MailAddr := '"';
NbDest := 0;
FOR KK := 1 TO CstNbUser DO
	IF AX_Subscribed[KK] AND AX_MailAddr[KK] <> '' AND (AX_User_LVL[KK] AND Fifo.out.Alarms_LVL)>0 THEN		// If user is subscribed to this alarm, add his mail adress to the list. 
		IF MailAddr = '"' THEN
			MailAddr := concat('"', AX_MailAddr[KK]);	// Initialize first sender. 
		END_IF
		NbDest := NbDest + 1;
	END_IF
END_FOR

IF NbDest >0 THEN
	IF NbDest>1 THEN
		FOR KK := 1 TO CstNbUser DO
			IF AX_Subscribed[KK] AND MailAddr <> AX_MailAddr[KK] AND (AX_User_LVL[KK] AND Fifo.out.Alarms_LVL)>0 THEN
				MailAddr := concat(concat(MailAddr, ', '), AX_MailAddr[KK]);		// append other mail adress if several users subsribed to this alarm. 
			END_IF
		END_FOR
	END_IF
	MailAddr := concat(MailAddr, '" ');
	bSendMail := TRUE;
	bAlarmNoDestinator	:= FALSE;
ELSE 
	bAlarmNoDestinator	:= TRUE;
	bSendMail 			:= FALSE;

END_IF	

SendMail
(
	NETID := ParamNetID,
	PATHSTR := concat(IN_Directory, 'SMTP.exe'),
	DIRNAME := IN_Directory,
	COMNDLINE := concat(str1 := MailAddr, str2 := body),
	start := bSendMail AND bWriteParam and not TON_Retry.Q
);

IF OUT_Completed THEN 
	SendMail(start := FALSE);
	OUT_Completed := FALSE;
	OUT_NbMailSent := OUT_NbMailSent + 1;

	bSendMail := FALSE;
	FIFO.A_Remove();
END_IF	

IF OUT_NbMailSent > 30000 THEN
	OUT_NbMailSent := 0;
END_IF

METHOD M_AlarmManager
VAR
	
	FB_AlarmCodeManager : FB_AlarmCodeManager;

END_VAR
// Gestion des alarmes internes au code

RS_AlarmDestinator(SET:= bAlarmNoDestinator , RESET1:= IN_Reset_OPC ) ; 

FB_AlarmCodeManager
(
	bAlarm1 := RS_AlarmDestinator.Q1,			// No recipient for at least one alarm
	bAlarm2 := OUT_Error,						// Out Error to send mail
	bAlarm3 := SendMail.ERR,					// Execution of SenMail.exe did not work. 
	bAlarm4 := FIFO.bOverwrite,					// Fifo Overflow
	bAlarm5 :=FALSE,							//
	bAlarm6 :=FALSE,    						//
	bAlarm7 :=FALSE,    						//
	bAlarm8 :=FALSE,    						//
	bAlarm9 :=FALSE,    						//
	bAlarm10 :=FALSE,   						//
	bAlarm11 :=FALSE,   						//
	bAlarm12 :=FALSE,   						//
	bAlarm13 :=FALSE,   						//
	bAlarm14 :=FALSE,   						//
	bAlarm15 :=FALSE,							//	
	wAlarmCode =>MesData.MesAlarmCode
);
END_METHOD

METHOD M_Evaluate
VAR 
END_VAR

Mesdata.AX_MailAddr		:= AX_MailAddr			;
Mesdata.AX_Subscribed	:= AX_Subscribed	    ;
MesData.AX_NomUtili		:= AX_NomUtili		    ;
MesData.OUT_NbMailSent	:= OUT_NbMailSent		;
MesData.AX_UserLVL		:= AX_User_LVL		    ;
END_METHOD

METHOD M_Init : BOOL
VAR_INPUT
END_VAR
END_METHOD

METHOD M_OPC : BOOL
VAR

END_VAR
Trig_OPC(CLK := IN_ChangePhoneMailInfos_OPC);
RS_OPC(SET:= Trig_OPC.Q);

//TrigRestartService(CLK := IN_Restart_Service_OPC);
//FUN_RestartStunnel(IN_Start := TrigRestartService.Q, IN_Directory := IN_Directory);


IF RS_OPC.Q1 THEN
	// Numéro de téléphone
	AX_MailAddr := OpcUa.AllValueW.AX_MailAddr_OPC;
	
	// Nom d'utilisateur
	AX_NomUtili	:= OpcUa.AllValueW.AX_NamesUsers_OPC;
	
	// User LVL . 
	AX_User_LVL := OpcUa.AllValueW.AX_UserLVL;
	
	// Mise a jour de la liste des subscribed
	AX_Subscribed := OpcUa.AllValueW.AX_SubscribedMail_OPC;

	RS_OPC(RESET1:= TRUE);
	RS_OPC(Reset1 := FALSE);
END_IF

Trig_Reset(CLK := IN_Reset_OPC);
IN_Reset_OPC := Trig_Reset.Q;
END_METHOD

METHOD M_Reset : BOOL
VAR_INPUT
END_VAR
VAR
	

END_VAR
FIFO.A_Reset();
IN_Reset_OPC 			:= FALSE;
bAlarmNoDestinator 		:= FALSE ;	
bSendMail				:= FALSE;
SendMail(Start:= FALSE ) ;
END_METHOD

END_PROGRAM

// ---- 04_Application/Annexes_Functions/PRG_AnnexesFunctions.TcPOU
PROGRAM PRG_AnnexesFunctions
VAR_INPUT PERSISTENT
	ParamServiceName_HH			: STRING(255) := 'RestartHH_CollectOR exe';	(*OPC UA Service Name*)
	ParamServiceName_OPCUA			: STRING(255) := 'OPCUA';	(*OPC UA Folder Name*)
	//ParamServiceName_Docker			: STRING(255) := 'dockerd';	(*Docker Service Name*)
	ParamServiceName_OpenVPN		: STRING(255) := 'OpenVPN';	(*OpenVPN folder  Name*)
	//ParamServiceName_Codesys		: STRING(255) := 'codesys3';	(*Codesys Service Name*)
	ParamServiceName_HMIServer		: STRING(255) := '';	(*OpenVPN UA Service Name*)	
	ParamServiceName_Teamviewer		: STRING(255) := 'Teamviewer';	(* Teamviewer Folder Name*)	
	
END_VAR
VAR_INPUT
	IN_bStartPing				: BOOL;	
    IN_bStart_IP				: BOOL;
    IN_bStart_PLC				: BOOL;

	IN_CmdRestart_HH			: BOOL;	// OPC UA , Docker , OPEn VPN , Codesys. Push button
	IN_CmdRestart_OPCUA 		: BOOL;	// OPC UA , Docker , OPEn VPN , Codesys. Push button
	IN_CmdRestart_OpenVPN 		: BOOL;	// OPC UA , Docker , OPEn VPN , Codesys. Push button
	IN_CmdRestart_Teamviewer 	: BOOL;	// OPC UA , Docker , OPEn VPN , Codesys. Push button
	IN_CmdRestart_HMIServer 	: BOOL;	// OPC UA , Docker , OPEn VPN , Codesys. Push button
	IN_CmdRestart_Docker 		: BOOL;	// OPC UA , Docker , OPEn VPN , Codesys. Push button	
	IN_CmdRestart_Codesys 		: BOOL;	// OPC UA , Docker , OPEn VPN , Codesys. Push button

	IN_bStartVpnConnection		: BOOL;
	IN_bStopVpnConnection		: BOOL;
	IN_AdrIP					: STRING(50);
END_VAR

VAR_INPUT PERSISTENT
	ParamRestartTCHour			: WORD := 3;
	ParamRestartTCEnabled		: BOOL ; 
END_VAR

VAR PERSISTENT 
	RestartCounter 				: UINT;
END_VAR

VAR
		bInit					: BOOL := TRUE ; 
		PRG_RestartService		: ARRAY[1..4] OF FB_RestartService ; 
		StartProcess 			: NT_StartProcess;
		CpuUsage				: TC_CpuUsage;
		TON_ALarm				: TON ; // TON to inhibate alarmes during the first secondes after initailization 

		// Restart Twincta
		Step: INT;
		R_Trig_TP_IP			: R_TRIG;
		TC_Restart1				: TC_Restart;	
		TP_GetIPPublic			: TP;

END_VAR
VAR_OUTPUT 
	CPUUsage_PLC				: UDINT ; 
END_VAR

IF bInit THEN
	M_Init();
	///////// 
END_IF




// Get Public IP : 	Auto query every 10 minutes
	FUN_GetPublicIp(
		ParamNetID := CstNetAmsId_IndusPC ,
		IN_DirExe := 'C:\TwinCAT\Functions\Annex_Fonctions\GetPublicIp\',
		IN_CmdStart := IN_bStart_IP OR (CalLocalTimeStruct.wMinute MOD 10 = 0 AND CalLocalTimeStruct.wSecond = 0
	));

// Ping Host 	
//	FUN_PingHost(IN_bStart := IN_bStartPing, IN_PingAdr := IN_AdrIP, IN_DirBatLocation := 'C:\TwinCAT\Functions\Fonction_Com\Ping\');

// CHECK STATES
	// CPU Usage 	
		CpuUsage(NETID := '', Start := CalLocalTimeStruct.wSecond = 0, TMOUT := T#1S);
		CPUUsage_PLC := 	CpuUsage.USAGE ; 
		
	// Check Disk Space = planned task
	// Check Services = planned task
	// Network Scan = planned task
	
	// VPN Management
		FUN_ConnectVPN(IN_CmdStart := IN_bStartVpnConnection, IN_OpenVpnFile := GVL_BASE.ParamOpenVpnFile);
		FUN_DisconnectVPN(IN_CmdStart := IN_bStopVpnConnection);
		

// RESTART SERVICES 
	// Restart OPC UA  	

			PRG_RestartService[1](ParamNetID:='' , IN_Directory := CONCAT(STR1:='C:\TwinCAT\Functions\Annex_Fonctions\RestartService\',STR2:= ParamServiceName_OpenVPN), Start:= IN_CmdRestart_OpenVPN , IN_ServiceName := 'RestartService.exe');

			PRG_RestartService[2](ParamNetID:='' , IN_Directory := CONCAT(STR1:='C:\TwinCAT\Functions\Annex_Fonctions\RestartService\',STR2:= ParamServiceName_OPCUA), Start:= IN_CmdRestart_OPCUA , IN_ServiceName := 'RestartService.exe');
	
			PRG_RestartService[3](ParamNetID:='' , IN_Directory := CONCAT(STR1:='C:\TwinCAT\Functions\Annex_Fonctions\RestartService\',STR2:= ParamServiceName_Teamviewer), Start:= IN_CmdRestart_Teamviewer , IN_ServiceName := 'RestartService.exe');
	


	// Restart PLC 	
		PRG_RestartPlc(CmdRestart:= IN_bStart_PLC);
		
	// Restart Twincat at specified date and time to fix EL6614 issue 
		CASE Step OF
			0: //	
				IF CalLocalTimeStruct.wHour = ParamRestartTCHour AND CalLocalTimeStruct.wMinute = 0 AND (CalLocalTimeStruct.wSecond >= 0 AND CalLocalTimeStruct.wSecond <=  5) AND ParamRestartTCEnabled  THEN 
					Step := 1;
				END_IF
			1:
				TC_Restart1(
					RESTART:= TRUE, 
					TMOUT:= T#500MS );
					RestartCounter:=RestartCounter+1;
		END_CASE
	
// ALARMS	
	//Gestion des alarmes sur active configuration --> Alarme inhibées pendant 10s
	TON_ALarm(IN:= MAIN.OUT_CalRunningPLC_IO , PT:= T#10S) ; 

	IF TON_Alarm.Q THEN 
		FUN_Alarms(IN_Directory := ParamDirBaseStore);
	END_IF
	
	FUN_CreateDir_CSV(InDirectory := ParamDirBaseStore);
	FUN_Write_CSV	(InDirectory := ParamDirBaseStore);

	
// Interfaces // 	

ModbusTcp() ; 
//HMI();

METHOD M_Init : BOOL
VAR_INPUT
END_VAR

VAR
	KK: UINT;
	LL: UINT;
END_VAR
	// Add code activation to the alarms
	
	FUN_Alarms_CSV.FIFO.A_Get();
	FUN_Alarms_CSV.FIFO.A_Remove();	
	FUN_Alarms_CSV.FIFO.In.Message := 'Code Activation';
	FUN_Alarms_CSV.FIFO.In.TimeStamp_Act := SYSTEMTIME_TO_STRING(CalLocalTimeStruct);
	FUN_Alarms_CSV.FIFO.A_Add();
	
	InfluxDb_AlarmsManagement.IN_FIFO.A_Get();
	InfluxDb_AlarmsManagement.IN_FIFO.A_Remove();
	InfluxDb_AlarmsManagement.IN_FIFO.In.Message := 'Code Activation';
	InfluxDb_AlarmsManagement.IN_FIFO.In.TimeStamp_Act := SYSTEMTIME_TO_STRING(CalLocalTimeStruct);
	InfluxDb_AlarmsManagement.IN_FIFO.A_Add();	
	
	FUN_SendMail.FIFO.A_Get();
	FUN_SendMail.FIFO.A_Remove();
	FUN_SendMail.FIFO.In.Message := 'Code Activation';
	FUN_SendMail.FIFO.In.TimeStamp_Act := SYSTEMTIME_TO_STRING(CalLocalTimeStruct);
	FUN_SendMail.FIFO.A_Add();
	
	// Reinitialize all Alarms values 
	FOR KK := 1 TO CstNbAlarmCode DO
		FUN_Alarms.AX_MesAlarmCode[KK] := 0 ; 
		FOR LL:=0 TO 15 DO 
			FUN_Alarms.AX_Journal[KK][LL].Value := FALSE ;
		END_FOR 
	END_FOR
	
	bInit:= False ;
END_METHOD

END_PROGRAM

// ---- 00_FunctionsBlocks/Beckhoff/Annexesfunction/FB_RestartService.TcPOU
FUNCTION_BLOCK FB_RestartService
VAR_INPUT
	IN_Directory			: T_MaxString; // directory of the file to compress
	ParamNetID				: STRING ; // Net ID of the PC with HH collector
	IN_ServiceName			: STRING  ;
	Start					: BOOL;
END_VAR
VAR
	StartProcess 			: NT_StartProcess;
	TrigStart				: R_TRIG;
END_VAR

TrigStart(CLK:=Start);
	StartProcess
	(
		NETID := ParamNetID,
		PATHSTR := concat(str1:= IN_Directory, str2 := IN_ServiceName),
		DIRNAME := IN_Directory,
		COMNDLINE := '',
		Start := TrigStart.Q,
		TMOUT := T#3M
	);
	IF NOT StartProcess.BUSY THEN
		IF NOT StartProcess.ERR THEN
			StartProcess(Start := FALSE);
		ELSE
			StartProcess(Start := FALSE);
		END_IF
	END_IF

END_FUNCTION_BLOCK

// ---- 04_Application/BDD/FUN_Write_CSV.TcPOU
PROGRAM FUN_Write_CSV
Var
    WriteValue          : FB_Write_CSV;
END_VAR
VAR_INPUT
 InDirectory             : T_MaxString;
AX_Variables            : ARRAY [1..500] OF ST_ValuesWrite;
END_VAR


WriteValue(InDirectory := InDirectory, ParamNbColumns := 36,AX_StructureValues := AX_Variables);

END_PROGRAM

// ---- 00_FunctionsBlocks/Beckhoff/DataProcessing/WriteFile/FB_Write_CSV.TcPOU
FUNCTION_BLOCK FB_Write_CSV
VAR_INPUT
	InDirectory 		: T_MaxString;
	AX_StructureValues	: ARRAY[1..500] OF ST_ValuesWrite;
	
	ParamNbColumns		: UINT := 200; 				(* (NA) Number of columns of the file*)
	ParamSeparateur		: STRING := ';';			(* (NA) Separator*)
	ParamDec			: STRING := ',';			(* (NA) ParamDec*)
	ParamExtension		: T_MaxString := '.csv'; 	(* (NA) csv extension *)
END_VAR
VAR_OUTPUT
END_VAR
VAR
	
    CompressFile        : FB_CompressFile;

MesData		: LoggerCSV;
	bWriteAlarm			: BOOL;						// Writing CSV File failed 
	TON_WritealarmFile	: TON;	
	// Data processing 
	format_string		: FB_FormatString;
	AX_AverageFunctions	: ARRAY[1..1000] OF FB_Average;
	AX_AverageValues	: ARRAY[1..1000] OF REAL;
	LenStringToWrite	: INT;
	
	GetHostName			: FB_GetHostName;
	CalFileName			: STRING;
	CalFileName_Old		: STRING;
	CalDate				: STRING;
	CalDate_Old			: STRING;
	
	//Test existence file 

	bFileOK				: BOOL := TRUE ;
	bDirChange			: BOOL;
	FindFile 			: FB_EnumFindFileEntry ;
	FileInfo			: ST_FindFileEntry;
	
	//Initial File creation 
	InitLine			: T_MaxString;
	LastInitLine		: T_MaxString;
	WelcomeMessage 		: T_MaxString := 'Daily rawdata file';
	ForDay				: T_MaxString := 'for day : ';
	ForPlant	 		: T_MaxString := 'for plant : ';
	NewLineVar			: T_MaxString := '$N';
	TimeStampVar		: T_MaxString := 'TimeStamp';
	len_to_write		: INT;
	len_to_add			: INT;
	
	WriteFileInit		: FB_WriteFile;
	WriteFile			: FB_WriteFile;
	MessageInitial		: ARRAY[1..100] OF T_Maxstring;
	MessageInitialNull	: ARRAY[1..100] OF T_Maxstring;
	bInitWrite			: BOOL;
	bInitWriting		: BOOL;
	
	// Write File
	LineToWrite			: ARRAY [1..100] OF  T_Maxstring;
	LineToWrite_Null	: ARRAY [1..100] OF  T_Maxstring;
	ValueToWrite		: T_MaxString;
	TriggerSampling		: R_TRIG;
	
	// General variables
	KK: UINT;
	bInit : BOOL;
	MesTimeStamp : STRING(19);
	

	
END_VAR

M_AlarmManager();
M_DataProcessing ();

IF NOT bInit THEN
	GetHostName(bExecute := FALSE);
	GetHostName(bExecute := TRUE);
	bInit := TRUE;
END_IF

format_string(
	sFormat := 'RAWDATA_%0.2d-%0.2d-%0.2d%s', 
	arg1 := F_WORD(in:=CalLocalTimeStruct.wYear),	arg2 := F_WORD(in:=CalLocalTimeStruct.wMonth),	arg3 := F_WORD(in:=CalLocalTimeStruct.wDay),
	arg4 := F_STRING(in:=ParamExtension),
	sOut => CalFileName
);

format_string(
	sFormat := '%0.2d-%0.2d-%0.2d', 
	arg1 := F_WORD(in:=CalLocalTimeStruct.wYear),	arg2 := F_WORD(in:=CalLocalTimeStruct.wMonth),	arg3 := F_WORD(in:=CalLocalTimeStruct.wDay),
	sOut => CalDate
);

format_string(
	sFormat := '%0.2d-%0.2d-%0.2d %0.2d:%0.2d:%0.2d', 
	arg1 := F_WORD(in:=CalLocalTimeStruct.wYear),	arg2 := F_WORD(in:=CalLocalTimeStruct.wMonth),	arg3 := F_WORD(in:=CalLocalTimeStruct.wDay),
	arg4 := F_WORD(in:=CalLocalTimeStruct.wHour),	arg5 := F_WORD(in:=CalLocalTimeStruct.wMinute),	arg6 := F_WORD(in:=CalLocalTimeStruct.wSecond),
	sOut => MesTimeStamp
);

InitLine := concat(str1:=WelcomeMessage, STR2:= concat(str1:=
	ParamSeparateur, str2:=concat(STR1:=ForDay, STR2:=concat(str1:= ParamSeparateur, STR2:= concat(str1:= 
	CalDate,str2:=concat(str1:= ParamSeparateur, str2 := CONCAT(str1:=
	ForPlant,str2:=Concat(str1:=ParamSeparateur, str2:= CONCAT(str1:= GetHostName.sHostName, str2:=ParamSeparateur)
))))))));

IF InitLine <> LastInitLine OR InitLine = '' OR (NOT FindFile.bError AND NOT bFileOK) THEN
	LastInitLine := InitLine;
	bInitWriting := TRUE;
END_IF
	
IF FUN_CreateDir_CSV.bDirOK THEN
	FindFile
	(
		sNetId := '',
		sPathName := concat(FUN_CreateDir_CSV.AX_DirNames[2],CalFileName),
		eCmd := eEnumCmd_First,
		bExecute := TRUE,
		tTimeout := T#3S,
		stFindFile => FileInfo
	);
	
MesData.TimeCreation 	:= FILETIME_TO_SYSTEMTIME(filetime := FileInfo.creationTime);
MesData.TimeModif	 	:= FILETIME_TO_SYSTEMTIME(filetime := FileInfo.lastWriteTime);
MesData.FileSize  		:= ULARGE_TO_ULINT(in := FileInfo.fileSize);	
	
	IF NOT FindFile.bBusy THEN
		FindFile(bExecute := FALSE);
		bFileOK := MesData.FileSize > 0 ; 
	END_IF
	
	IF FindFile.bError OR  NOT bFileOK THEN
		FUN_CreateDir_CSV(InDirectory := ParamDirBaseStore, RESET2 := TRUE);
	END_IF
	
	IF NOT FindFile.bBusy AND NOT bFileOK AND bInitWriting THEN
		// je réinitialise les longueurs
		len_to_write := 0;
		MessageInitial := MessageInitialNull;
		MEMCPY(destAddr := ADR(MessageInitial)+len_to_write, srcAddr := ADR(InitLine), n := len(InitLine));
		len_to_add := len(InitLine);			len_to_write := len_to_write + len_to_add;
		
		MEMCPY(destAddr := ADR(MessageInitial)+len_to_write, srcAddr := ADR(NewLineVar), n := len(NewLineVar));
		len_to_add := len(NewLineVar);			len_to_write := len_to_write + len_to_add;
		
		MEMCPY(destAddr := ADR(MessageInitial)+len_to_write, srcAddr := ADR(TimeStampVar), n := len(TimeStampVar));
		len_to_add := len(TimeStampVar);		len_to_write := len_to_write + len_to_add;
		
		MEMCPY(destAddr := ADR(MessageInitial)+len_to_write, srcAddr := ADR(ParamSeparateur), n := len(ParamSeparateur));
		len_to_add := len(ParamSeparateur);		len_to_write := len_to_write + len_to_add;
		
		FOR KK := 1 TO ParamNbColumns DO
			MEMCPY(destAddr := ADR(MessageInitial)+len_to_write, srcAddr := ADR(AX_StructureValues[KK].Description), n := len(AX_StructureValues[KK].Description));
			len_to_add := len(AX_StructureValues[KK].Description);			len_to_write := len_to_write + len_to_add;
			
			MEMCPY(destAddr := ADR(MessageInitial)+len_to_write, srcAddr := ADR(ParamSeparateur), n := len(ParamSeparateur));
			len_to_add := len(ParamSeparateur);								len_to_write := len_to_write + len_to_add;
		END_FOR
		
		MEMCPY(destAddr := ADR(MessageInitial)+len_to_write, srcAddr := ADR(NewLineVar), n := len(NewLineVar));
		len_to_add := len(NewLineVar);			len_to_write := len_to_write + len_to_add;
		
		WriteFileInit
		(
			InStart := TRUE,
			InDirFile := concat(FUN_CreateDir_CSV.AX_DirNames[2], CalFileName),
			InAmsId := '', 
			InPMessage := ADR(MessageInitial),
			InLMessage := len_to_write
		);
		
		IF WriteFileInit.OutCompleted OR bFileOK THEN
			WriteFileInit(InStart := FALSE);
		END_IF
	END_IF
	
	
	// Write file on SampleRate
	
	TriggerSampling(clk := CalLocalTimeStruct.wSecond = 10);

	IF bFileOK AND MesData.FileSize < 100000000  THEN
		bInitWriting := FALSE;
		len_to_write := 0;
		LineToWrite := LineToWrite_Null;
		MEMCPY(destAddr := ADR(LineToWrite)+len_to_write, srcAddr := ADR(MesTimeStamp), n := len(MesTimeStamp));
		len_to_add := len(MesTimeStamp);		len_to_write := len_to_write + len_to_add;
		
		MEMCPY(destAddr := ADR(LineToWrite)+len_to_write, srcAddr := ADR(ParamSeparateur), n := len(ParamSeparateur));
		len_to_add := len(ParamSeparateur);		len_to_write := len_to_write + len_to_add;
		
		FOR KK := 1 TO ParamNbColumns DO
			ReplaceAll(IN_StringToSearch := REAL_TO_STRING(AX_AverageValues[KK]), IN_StringToFind := '.', IN_StringToReplace := ParamDec, OUT_StringToSearch => ValueToWrite);
			//ValueToWrite := REAL_TO_STRING(AX_AverageValues[KK]);
			MEMCPY(destAddr := ADR(LineToWrite)+len_to_write, srcAddr := ADR(ValueToWrite), n := len(ValueToWrite));
			len_to_add := len(ValueToWrite);	len_to_write := len_to_write + len_to_add;
			
			MEMCPY(destAddr := ADR(LineToWrite)+len_to_write, srcAddr := ADR(ParamSeparateur), n := len(ParamSeparateur));
			len_to_add := len(ParamSeparateur);	len_to_write := len_to_write + len_to_add;
		END_FOR
		MEMCPY(destAddr := ADR(LineToWrite)+len_to_write, srcAddr := ADR(NewLineVar), n := len(NewLineVar));
		len_to_add := len(NewLineVar);			len_to_write := len_to_write + len_to_add;
		
		WriteFile
		(
			InStart := TriggerSampling.Q,
			InDirFile := concat(FUN_CreateDir_CSV.AX_DirNames[2], CalFileName),
			InAmsId := '', 
			InpMessage := ADR(LineToWrite),
			InLMessage := len_to_write
		);
		
		IF NOT WriteFile.OutBusy AND NOT WriteFile.OutError AND WriteFile.OutCompleted THEN
			// File has been writen successfully
			bWriteAlarm	:= FALSE ;
		ELSIF WriteFile.OutError THEN 
			// In case of writing error, try again to write the alarm. 
			bWriteAlarm	:= TRUE ;
		
		END_IF		
		
	END_IF

END_IF

CompressFile(IN_Directory := InDirectory);

METHOD M_AlarmManager
VAR

	FB_AlarmCodeManager			: FB_AlarmCodeManager ;

END_VAR
TON_WritealarmFile(IN:= NOT bFileOK  , PT:= T#10S  ) ;

// ALARM CODE //
	FB_AlarmCodeManager(
		bAlarm1			:= bWriteAlarm	  ,				// Write CSV Alarm
		bAlarm2			:= FALSE   ,					// 
		bAlarm3			:= TON_WritealarmFile.Q   ,		// Can not create CSV Alarm file 
		bAlarm4			:= FALSE	 ,					//
		bAlarm5			:= FALSE	,					// 
		bAlarm6			:= FALSE,									//
		bAlarm7			:= FALSE,                                   //
		bAlarm8			:= FALSE,                                   //
		bAlarm9			:= FALSE,                                   //
		bAlarm10		:= FALSE,                                   //
		bAlarm11		:= FALSE,									//
		bAlarm12		:= FALSE,                                   //
		bAlarm13		:= FALSE,                                   //
		bAlarm14		:= FALSE,                                   //
		bAlarm15		:= FALSE,                                   //
		wAlarmCode		=>MesData.MesAlarmCode);
END_METHOD

METHOD M_DataProcessing : BOOL
VAR
		
	KK : UINT;
END_VAR
FOR KK := 1 TO ParamNbColumns DO 
	IF AX_StructureValues[KK].Address <> 0 THEN 	
		AX_AverageFunctions[KK](ValueIn := AX_StructureValues[KK].Address^, WindowDuration := AX_StructureValues[KK].Sampling, CycleTime := CstCycleTime_Annex, ValueOut=> AX_AverageValues[KK]);	
	ELSIF AX_StructureValues[KK].AddressLR <> 0 THEN 	
		AX_AverageFunctions[KK](ValueIn := AX_StructureValues[KK].AddressLR^, WindowDuration := AX_StructureValues[KK].Sampling, CycleTime := CstCycleTime_Annex, ValueOut=> AX_AverageValues[KK]);	
	ELSIF AX_StructureValues[KK].AddressUL <> 0 THEN 	
		AX_AverageFunctions[KK](ValueIn := AX_StructureValues[KK].AddressUL^, WindowDuration := AX_StructureValues[KK].Sampling, CycleTime := CstCycleTime_Annex, ValueOut=> AX_AverageValues[KK]);	
	ELSIF AX_StructureValues[KK].AddressUI <> 0 THEN
		AX_AverageFunctions[KK](ValueIn := AX_StructureValues[KK].AddressUI^, WindowDuration := AX_StructureValues[KK].Sampling, CycleTime := CstCycleTime_Annex, ValueOut=> AX_AverageValues[KK]);			
	ELSE
		AX_AverageValues[KK] := 0;
	END_IF
END_FOR
END_METHOD

END_FUNCTION_BLOCK

// ---- 00_FunctionsBlocks/Common/Ctrl/FB_PIDRegulation.TcPOU
FUNCTION_BLOCK FB_PIDRegulation
// Akuo Version of PID Regulation  for solar power plant . Input can be P or Q . 
// Out  = Error *K (1+ 1/Ti sum(error) + Td delta(error) ) 
(*
	DATE :						07/2020																										
	Developper:				GGY																												
	Version :					V1.0																										
	Function :																																																																		
*)
VAR_INPUT PERSISTENT

	ParamK				: REAL ; // Proportionnal 
	ParamTi				: REAL ; // Integral (s) . 0 to disable
	ParamTd				: REAL ; // Derivative (s). 0 to disable . 
	
	ParamXmax			: REAL ; // maximal Value for X. Shall account for number of available PTR . 
	ParamXmin			: REAL; // minimal value for X 
	
	ParamOutmax			: REAL ; // Maximal output value
	ParamOutmin			: REAL ; // Maximal input value 
	
	
	
END_VAR

VAR_INPUT
	IN_SetptX				: REAL ; // Value to reach 
	IN_MesX					: REAL ; // Measure to compare with
	IN_MesComXError			: BOOL ; // Communication lost with the measure tool. 
	IN_SetptOpenLoop		: REAL  ; // Output of the PID when disabled. This shall be equal to an evaluation of the correct output. Usually SetptX. OpenLoop setpoint. 

	
	IN_CmdReset				: BOOL ; // Reset PID 
	IN_CmdPIDOn				: BOOL ; // Activate/ Desactivate PID . outpout equals to the offset if desactivated/ 
END_VAR

VAR_OUTPUT
	OUT_X					: REAL ; // Output of the PID 
	OUT_PIDMode				: INT ; // Mode of the PID ( 1: Bypassed  , 3 : Proportionnal , 4 : PI , 5 PID , 6: PD). 
	
END_VAR
VAR
	
	CalSetptOffset 			: REAL  ; // Offset to be added to the PID to ensure continuity when resetting it or activating it. 

	IntegralX			: REAL ; // Intergal
	DerivativeX			: REAL ; // Derivative
	ErrorX				: REAL;	// Error  
	CP_PID				: BOOL;	// PID Enabled
	Clock				: TON ; // Calculate Elapsed Time ; 
	DeltaTime			: DWORD ; // 
	// Derivative
	StepDerivative		: INT := 0; // Derivative Step ( initialization , methode degre 1 , methode degre 2) 
	X2,X1				:REAL;
	T1					:DWORD;
	CalReset: BOOL;
	
	KCopy				: REAL ; 
	TiCopy				: REAL ; 
	TdCopy				: REAL ; 
	X_Temp				: REAL ; // Intermediate result . 
	
	CalOutLimitReached_Up	: BOOL;		// Output reached maximum output limit
	CalOutLimitReached_Down	: BOOL;		// Output reached minimum output limit
	
	TrigCP_PID: BOOL;
	bInit: BOOL := TRUE  ; 
	time_new: INT;
	delta_time: INT;
	time_old: INT;
END_VAR

// INITIALIZE 
	OUT_PIDMode := 1 ;

	CalReset := IN_CmdReset OR NOT IN_CmdPIDOn OR ABS(KCopy-ParamK)>0.000001 OR ABS(TiCopy-ParamTi)>0.000001 OR ABS(TdCopy-ParamTd)>0.000001 OR IN_MesComXError; // Reset if change of parameters >> passage en boucle ouverte. 

	CP_PID :=   (ParamK>0.00001 OR ParamK<-0.00001)  AND NOT CalReset  ; // PID Enable ssi Activation and K >0 and not communication alarm with power meter . and not K change . 
	

	IF NOT CP_PID OR bInit THEN 
		// Début proposition de modif KBT
		time_old := TIME_TO_INT(TIME());
		// Fin proposition de modif KBT

		
		Clock(IN:=FALSE ) ; 
		Clock(IN:=TRUE, PT:=T#1H);	//Initialize clock 
		bInit	:= FALSE ; 
	ELSE 
		Clock();
		DeltaTime	:= TIME_TO_DWORD(CLOCK.ET) ; 	// 
		
		// Début proposition de modif KBT
		time_new := TIME_TO_INT(TIME());
		IF time_old <> 0 THEN
			delta_time := time_new - time_old;
		END_IF
		time_old := TIME_TO_INT(TIME());
		// Fin proposition de modif KBT
	END_IF


	KCopy 	:=  ParamK ; 
	TiCopy	:= ParamTi ; 
	TdCopy	:= ParamTd ; 
	
// CHECK INPUT // 
	IN_SetptX := MAX(MIN(IN_SetptX, ParamXmax ), ParamXmin); // Limit the Input with Min/ Max values.

	IN_SetptOpenLoop := MAX(MIN(IN_SetptOpenLoop, ParamXmax ), ParamXmin); // Limit the Input with Min/ Max values.
	
// EVALUATE QUANTITIES //
	// Clock
	
	IF DeltaTime > 0 THEN	// We calculate on time cycle. When the time cycle is over , we reinitialize the clock
		Clock(IN:=FALSE ) ; 
		Clock(IN:=TRUE, PT:=T#1H);	//Initialize clock 
	ELSE
		CLOCK(PT:=T#1H,IN:=TRUE);
	END_IF
	// Error 
		ErrorX := IN_SetptX - IN_MesX ; 

	//Integral
		// Sauturate the integral if overflow or if limts are reached or output reaches limits Reset the integral if command reset. 
		IF (NOT(1E30 - ErrorX*DeltaTime/1000 < IntegralX OR -1E30 - ErrorX*DeltaTime/1000 > IntegralX) AND ParamTi>0 ) OR CalReset THEN
			IF NOT ((ErrorX > 0 AND  CalOutLimitReached_Up) OR (ErrorX < 0 AND CalOutLimitReached_Down)) THEN 
				IntegralX:=SEL(CalReset,IntegralX+ErrorX*DeltaTime/1000 , 0) ;
			END_IF
			
			
		END_IF
		
	// Derivative 
		IF StepDerivative=0 OR CalReset THEN		// Reinitializa derivative if reset commAND  
			X1:=ErrorX;
			X2:=ErrorX;
			T1:=DeltaTime;
			DerivativeX := 0;
			StepDerivative:=1;
		ELSIF StepDerivative=1 AND ParamTd>0 THEN 
			DerivativeX := (ErrorX - X1)/(DeltaTime-T1) ; // f'(x) = (f(x+h)-f(x))/h
			X2:=X1;
			X1:=ErrorX;
			T1:=DeltaTime;	
			StepDerivative:=2 ; 		
		ELSE	
			IF DeltaTime>0 AND DerivativeX < 1E30 AND DerivativeX> 1E30 AND ParamTd>0  THEN		// Saturate the derivative if going too high. 
				IF NOT ((ErrorX > 0 AND  CalOutLimitReached_Up) OR (ErrorX < 0 AND CalOutLimitReached_Down)) THEN 
					DerivativeX:=(3*(ErrorX)-4*X1+X2)/(2*(DeltaTime-T1)*1000);		// Formule de Gear au second degré . f'(x) = 1/2h*(3*f(x+2h)-4*f(x+h)+f(x))
					X2:=X1;
					X1:=ErrorX;
					T1:=DeltaTime;
				END_IF
			END_IF;
		END_IF;
	
// PID CALCULATION
	IF CP_PID THEN

		
		TrigCP_PID	:= TRUE ; 
		// PID Enable 
		IF  ParamTi>0 AND ParamTd>0 THEN // Integral and derivative activated
			X_Temp:=CalSetptOffset+ParamK*(ErrorX+IntegralX/ParamTi+DerivativeX*ParamTd);
			OUT_PIDMode := 5 ; 
		ELSIF ParamTd>0 THEN // Derivative activated 
			X_Temp:= CalSetptOffset+ParamK*(ErrorX+DerivativeX*ParamTd) ; 
			OUT_PIDMode := 6 ; 
		ELSIF ParamTi>0 THEN // Integral activated 
			X_Temp:=CalSetptOffset+ParamK*(ErrorX+IntegralX/ParamTi);
			OUT_PIDMode := 4 ; 
		ELSE	// Only proportionnal
			X_Temp:=CalSetptOffset+ParamK*(ErrorX) ; 
			OUT_PIDMode := 3 ; 
		END_IF
		
	ELSE
		
		CalSetptOffset := IN_SetptOpenLoop ; // At the moment when i activated the PID, i need to ensure continuity of the OUT_X and start the PID from there . 
	
		TrigCP_PID	:= FALSE ; 
		//PID Disable. Open Loop . 
		X_Temp := IN_SetptOpenLoop ;
		OUT_PIDMode:=1 ;
	END_IF
	
// Saturate the OUtput with limits : 
CalOutLimitReached_Up := (X_Temp > ParamOutmax)  ;
CalOutLimitReached_Down:= (X_Temp < ParamOutmin)  ;
 

OUT_X :=  MAX(MIN(ParamOutmax , X_Temp ) , ParamOutmin ) ;

END_FUNCTION_BLOCK

// ---- 01_Equipement_Library/Actuators/FB_CB_GridMVCB.TcPOU
FUNCTION_BLOCK FB_CB_GridMVCB EXTENDS FB_CB_Base
//////////////////
//  Motorized Circuit Breaker with telecommAND   Requires Open and Close impulsions.
//////////////////

VAR_INPUT PERSISTENT
	// Parameters of the Object (instance/model specific) 
	
END_VAR

VAR_INPUT
	// I/O Inputs              	
		
END_VAR

VAR
	//M_OPENCLOSE VARIABLES//

	
	//M_ALARMMANAGEMENT VARIABLES//
		
	//M_STATEMANAGER VARIABLES//
MesDataExd			: CB_Standard ; 
	// M_EXECUTE VARIABLES //
		
	

		
END_VAR

METHOD M_AlarmManagement
//////////////////
// Manages Contactor alarms and warnings
/////////////////

VAR 
	// Method local variables (reinitialized at each cycle) 
	FB_AlarmCodeManager			: FB_AlarmCodeManager ; 

	
END_VAR
VAR_INPUT
	
END_VAR
// Check if command and measures are matching after tempo
TON_NotClosedAndNotOpened(IN:=  NOT MesClosed AND NOT MesOpened , PT := ParamTimeOut_Alarm) ; 
TON_ClosedAndOpened(IN:= MesClosed AND MesOpened, PT := ParamTimeOut_Alarm) ; 
//RS_AlarmStopReclose(Set := MesTransfo_Fault, RESET1 := BlockWriteTemp[1] OR IN_CmdReset_L);

// ALARM CODE //
	FB_AlarmCodeManager(
		bAlarm1			:= FALSE, 									// 
		bAlarm2			:= TON_NotClosedAndNotOpened.Q,				// Incoherent State mesure (Not Opened and not Closed )
		bAlarm3 		:= TON_ClosedAndOpened.Q,	 				// Incoherent State mesure (Opened and Closed )	
		bAlarm4			:= FALSE, 									// 
		bAlarm5			:= FALSE, 									//
		bAlarm6			:= FALSE,                                   //
		bAlarm7			:= FALSE,                                   //
		bAlarm8			:= FALSE,                                   //
		bAlarm9			:= FALSE,                                   //
		bAlarm10		:= FALSE,                                   //
		bAlarm11		:= FALSE,                                   //
		bAlarm12		:= FALSE,                                   //
		bAlarm13		:= FALSE, 									//
		bAlarm14		:= FALSE, 									//
		bAlarm15		:= FALSE, 									// 
		wAlarmCode		=>MesDataExd.MesData.MesAlarmCode);

//WARNING CODE //
		FB_AlarmCodeManager(
		bAlarm1			:= FALSE, 									//
		bAlarm2			:= FALSE,	 		                        //
		bAlarm3 		:= FALSE,									//		
		bAlarm4			:= FALSE, 									//
		bAlarm5			:= FALSE,                                   //
		bAlarm6			:= FALSE,                                   //
		bAlarm7			:= FALSE,                                   //
		bAlarm8			:= FALSE,                                   //
		bAlarm9			:= FALSE,                                   //
		bAlarm10		:= FALSE,                                   //
		bAlarm11		:= FALSE,                                   //
		bAlarm12		:= FALSE,                                   //
		bAlarm13		:= FALSE,                                   //
		bAlarm14		:= FALSE,                                   //
		bAlarm15		:= FALSE,                                   //
		wAlarmCode 		=>MesDataExd.MesData.MesWarningCode);

// EVENT CODE //
	FB_AlarmCodeManager(
		bAlarm1			:= FALSE, 									// 
		bAlarm2			:= FALSE, 									// 
		bAlarm3			:= MesOpened, 								// Opened Position
		bAlarm4			:= MesClosed, 								// Closed Position
		bAlarm5			:= IN_CmdReset_L,                           // Reset Command
		bAlarm6			:= FALSE,                                   //
		bAlarm7			:= FALSE,                                   //
		bAlarm8			:= FALSE,                                   //
		bAlarm9			:= FALSE,                                   //
		bAlarm10		:= FALSE,                                   //
		bAlarm11		:= FALSE,                                   //
		bAlarm12		:= FALSE,                                   //
		bAlarm13		:= FALSE,                                   //
		bAlarm14		:= FALSE,                                   //
		bAlarm15		:= FALSE,                                   //
		wAlarmCode		=>MesDataExd.MesData.MesEventCode);
END_METHOD

METHOD M_Execute
VAR_INPUT
END_VAR
// PERMANENT CONDITIONS //	
MesDataExd.MesData.MesCP_Open					:= IN_CmdOpen AND NOT IN_CmdReset_L;
MesDataExd.MesData.MesCP_Close				:= NOT MesDataExd.MesData.MesClosed AND IN_CmdClose AND NOT MesDataExd.MesData.MesAlarmCode.0 AND NOT MesDataExd.MesData.MesCP_Open AND NOT IN_CmdReset_L ;



SUPER^.M_Execute();
END_METHOD

METHOD M_StateManager
//////////////////
// Manages Contactor State
/////////////////

VAR 
	// Method local variables (reinitialized at each cycle) 
	
END_VAR
MesState := 0 ; 
IF MesOpened THEN		// If the cell seems opens and closed in the same time, we will consider it as opened. 
	
	MesState.0 := 1 ; 
MesDataExd.MesData.MesClosed := FALSE ; 
MesDataExd.MesData.MesOpened := TRUE ; 
ELSIF MesClosed THEN
	
	MesState.1 := 1 ; 
MesDataExd.MesData.MesClosed := TRUE ; 
MesDataExd.MesData.MesOpened := FALSE ; 
ELSE 
	MesState.0 := 1 ;		// if the cell seems neither opened and neither closed , we will consider it as opened. 
MesDataExd.MesData.MesClosed := FALSE ; 	
MesDataExd.MesData.MesOpened := TRUE ; 
END_IF
END_METHOD

END_FUNCTION_BLOCK

// ---- 01_Equipement_Library/Actuators/FB_CB_Base.TcPOU
FUNCTION_BLOCK FB_CB_Base
//////////////////
// Electrical Switch - Base FB
//////////////////

VAR_INPUT PERSISTENT
	// Parameters of the Object (instance/model specific) 
	ParamTimeOut_Open       		: TIME  := T#1S     ;       (* (ms) Config : Tempo to open before Timeout warning  *)
	ParamTimeOut_Close      		: TIME  := T#1S     ;		(* (ms) Config : Tempo to close before Timeout warning*)
	ParamTimeOut_Alarm   		    : TIME  := T#200MS  ;		(* (ms) Config : Tempo when open and close before raising alarm*)
	ParamNC							: BOOL  := FALSE    ;		(* (NA) False: TRUE = Closed, True : TRUE = opened*)
	ParamNbFdbck			    	: BYTE  := 1        ;		(* (NA) Number of feedback position (1: 1 wire, 2 : 2 wire)*)
	ParamClosedInput_Connected		: BOOL  := TRUE     ; 		(* (NA) True : closed input is connected*)
	                                                    	
END_VAR

VAR_OUTPUT
	//Child objects
	
END_VAR

VAR_INPUT
	// I/O Inputs 
		IN_MesOpened_IO					: BOOL  ; 				// (NA) [P,H,B] Opened Position IO	         
		IN_MesClosed_IO 				: BOOL := TRUE ; 		// (NA) [P,H,B] Closed Position IO           
	
		IN_CmdOpen 						: BOOL ; 				// (NA) External Open Command 
		IN_CmdClose						: BOOL ; 				// (NA) External Close Command 
		
	{attribute 'OPC.UA.DA' := '1'}   
		IN_CmdReset_L					: BOOL ;				// (NA) External Reset Command              // Check: what does the L respresent ? 
END_VAR

VAR
	//M_OPENCLOSE VARIABLES//
		MesOpened					     : BOOL ;                                                                     
		MesClosed					     : BOOL ;                                                                     
		
	//M_ALARMMANAGEMENT VARIABLES//
		FB_CheckCommand				     : FB_CheckCommand ; 	//(NA) Check if start command successful 
		FB_CheckCommand2			     : FB_CheckCommand ;	//(NA) Check if stop command successful  
		TON_ClosedAndOpened			     : TON ;              	
		TON_NotClosedAndNotOpened	     : TON ;              	
                                             	
		
		
	//M_STATEMANAGER VARIABLES//
		MesState					     : BYTE ; 				// (NA) Cal [P,H,B] Bit 0: Open , Bit 1: Closed        
	///MesDataExd				     : CB ; 

	// M_EXECUTE VARIABLES 	//                                   
		MesCP_Open		: BOOL ;   	(* Cal(NA) Permanent Conditions*)
		MesCP_Close		: BOOL ; 	(* Cal(NA) Permanent Conditions*) 

		
END_VAR

METHOD M_AlarmManagement
//////////////////
// Manages Contactor alarms and warnings
/////////////////

VAR 
	// Method local variables (reinitialized at each cycle) 

	
END_VAR
END_METHOD

METHOD M_Execute
VAR_INPUT
END_VAR
// If One wire feedback , Open Position is the inverse of Close Position. 
	IF  ParamNbFdbck=1 AND ParamClosedInput_Connected THEN
		IN_MesOpened_IO := NOT IN_MesClosed_IO ;
	ELSIF ParamNbFdbck = 1 AND NOT ParamClosedInput_Connected THEN
		IN_MesClosed_IO := NOT IN_MesOpened_IO;
	END_IF
	
	IF ParamNC THEN 
		MesOpened := NOT IN_MesOpened_IO ; 
		MesClosed := NOT IN_MesClosed_IO ; 
	ELSE
		MesOpened := IN_MesOpened_IO ; 
		MesClosed := IN_MesClosed_IO ; 		
	END_IF
	
	
//Methods call	
	M_OpenClose(); 
	M_StateManager() ;
	M_AlarmManagement();
END_METHOD

METHOD M_OpenClose
//////////////////
// Manages Opening of the contactor
//////////////////

VAR 
	// Method local variables (reinitialized at each cycle) 
	
END_VAR
END_METHOD

METHOD M_StateManager
//////////////////
// Manages Contactor State
/////////////////

VAR 
	// Method local variables (reinitialized at each cycle) 
	
END_VAR
END_METHOD

END_FUNCTION_BLOCK

// ---- 01_Equipement_Library/Actuators/FB_CB_MainHVCB.TcPOU
FUNCTION_BLOCK FB_CB_MainHVCB EXTENDS FB_CB_Base
//////////////////
//  Motorized Circuit Breaker with telecommAND  Requires Open and Close impulsions.
//////////////////

VAR_INPUT PERSISTENT
	// Parameters of the Object (instance/model specific) 
	ParamTP_Impulsion		    : TIME 		:= T#2S ;	(* (s) Config : Tempo for the start or stop command impulsion											*)
	ParamComutNc			    : BOOL ;                (**)
	ParamSectLigne			    : BYTE      :=1 ;		(* (NA) Monitoring du sectionneur de ligne de la MainMVCB.0 = TRUE := Monitoré .1 = TRUE Close is connected, .2 = ParamNC*)

END_VAR

VAR_OUTPUT
	//Child objects
	
END_VAR

VAR_INPUT
	A1_Sect				       : FB_CB_MVSwitch;

// I/O Inputs              
	IN_MesAlarmPwr_IO		           : BOOL ;	              // (NA)[P,H,B] Remote control Power supply Error .  IO  	
	IN_MesTripped_IO		  		   : BOOL ; 	          // Tripped position of the CB Must Ack To switch in again
	IN_MesComut_IO			   	   : BOOL := TRUE ; 	  // True if cell is in local position . 
	IN_MesEarth_IO 			       : BOOL ; 	
		
END_VAR

VAR
	//M_OPENCLOSE VARIABLES//	
	TP_Open	 			: TP ;				// (NA) Temporisation for Open pulse Command
	TP_Close 				: TP ;				// (NA) Temporisation for Close pulse Command	

	//M_ALARMMANAGEMENT VARIABLES//
MesDataExd	        :  CB_MainHVCB_Sch ; 
	
//M_STATEMANAGER VARIABLES//
	
END_VAR

METHOD M_AlarmManagement
//////////////////
// Manages Contactor alarms and warnings
/////////////////

VAR 
	// Method local variables (reinitialized at each cycle) 
	FB_AlarmCodeManager			: FB_AlarmCodeManager ; 
	
	CmdOpenCloseIO: BOOL; //Check IN/OUT_CMDOpenClose
END_VAR


TON_NotClosedAndNotOpened(IN:=  NOT MesClosed AND NOT MesOpened , PT := ParamTimeOut_Alarm) ; 
TON_ClosedAndOpened(IN:=MesClosed AND MesOpened, PT := ParamTimeOut_Alarm) ; 


// ALARM CODE //
	FB_AlarmCodeManager(
		bAlarm1			:= MesDataExd.MesTripped,					// Cb is tripped
		bAlarm2			:= TON_NotClosedAndNotOpened.Q,				// Incoherent State mesure (Not Opened and not Closed )
		bAlarm3 		:= TON_ClosedAndOpened.Q   , 				// Incoherent State mesure (Opened and Closed )	
		bAlarm4			:= FALSE, 				// 
		bAlarm5			:= FALSE  , 			// 
		bAlarm6			:= FALSE,                                   //
		bAlarm7			:= FALSE,                                   //
		bAlarm8			:= FALSE,                                   //
		bAlarm9			:= FALSE,                                   //
		bAlarm10		:= FALSE,                                   //
		bAlarm11		:= FALSE,                                   //
		bAlarm12		:= FALSE,                                   //
		bAlarm13		:= FALSE,                                   //
		bAlarm14		:= FALSE,                                   //
		bAlarm15		:= FALSE , 									//
		wAlarmCode		=>MesDataExd.MesData.MesAlarmCode);

//WARNING CODE//
		FB_AlarmCodeManager(
		bAlarm1			:= FALSE,//
		bAlarm2			:= FALSE,//
		bAlarm3 		:= FALSE,										// 
		bAlarm4			:= MesDataExd.MesAlarmPwr, 						// Power Supply Fault
		bAlarm5			:= MesDataExd.MesComutLocal, 					// COMUTATUTOR IN LOCAL
		bAlarm6			:= MesDataExd.MesEarth, 							// Earthing is done 
		bAlarm7			:= SEL( ParamSectLigne.0 ,FALSE ,  NOT A1_Sect.MesDataExd.MesData.MesClosed),				// Sectionneur de ligne ouvert 
		bAlarm8			:= FALSE, 										//
		bAlarm9			:= FALSE,                                       //
		bAlarm10		:= FALSE,                                       //
		bAlarm11		:= FALSE,                                       //
		bAlarm12		:= FALSE,                                       //
		bAlarm13		:= FALSE,                                       //
		bAlarm14		:= FALSE,                                       //
		bAlarm15		:= FALSE, 										//
		wAlarmCode 		=>MesDataExd.MesData.MesWarningCode);

// EVENT CODE //
	FB_AlarmCodeManager(
		bAlarm1			:= FALSE, 			// 
		bAlarm2			:= FALSE, 		    // 
		bAlarm3			:= MesOpened, 				// Opened Position
		bAlarm4			:= MesClosed, 				// Closed Position
		bAlarm5			:= IN_CmdReset_L, 			// Reset command
		bAlarm6			:= FALSE, 					//
		bAlarm7			:= FALSE,                   //
		bAlarm8			:= FALSE,                   //
		bAlarm9			:= FALSE,                   //
		bAlarm10		:= FALSE,                   //
		bAlarm11		:= FALSE,                   //
		bAlarm12		:= FALSE,                   //
		bAlarm13		:= FALSE, 					//
		bAlarm14		:= FALSE,                   //
		bAlarm15		:= FALSE,                   //
		wAlarmCode		=>MesDataExd.MesData.MesEventCode);   
		                                            
	//                                              
	                                                
	// UPDATE STRUCTURE

	IF ParamComutNc THEN
	MesDataExd.MesComutLocal	:= NOT IN_MesComut_IO ; 
	ELSE
	MesDataExd.MesComutLocal	:= IN_MesComut_IO ; 
	END_IF
	
MesDataExd.MesAlarmPwr		    := IN_MesAlarmPwr_IO ; 
MesDataExd.MesTripped			:= IN_MesTripped_IO ; 
MesDataExd.MesEarth			    := IN_MesEarth_IO ; 
MesDataExd.MesOpened_Sect	        := SEL(ParamSectLigne.0 , FALSE  , NOT A1_Sect.MesDataExd.MesData.MesClosed ) ;
END_METHOD

METHOD M_Execute
VAR_INPUT
END_VAR

VAR

END_VAR
//MainMVCB avec etat de sectionneur de ligne
IF ParamSectLigne.0 THEN 
	A1_Sect.ParamNbFdbck := 1;
	A1_Sect.ParamNC := ParamSectLigne.2;
	A1_Sect.ParamClosedInput_Connected := ParamSectLigne.1 ; 
	A1_Sect.M_Execute();
END_IF

// PERMANENT CONDITIONS //	
MesDataExd.MesData.MesCP_Open					:= IN_CmdOpen AND NOT IN_CmdReset_L;
MesDataExd.MesData.MesCP_Close				:= NOT MesDataExd.MesData.MesClosed AND IN_CmdClose AND NOT MesDataExd.MesData.MesAlarmCode.0 AND NOT MesDataExd.MesData.MesCP_Open AND NOT IN_CmdReset_L ;


SUPER^.M_Execute();
END_METHOD

METHOD M_StateManager
//////////////////
// Manages Contactor State
/////////////////

VAR 
	// Method local variables (reinitialized at each cycle) 
	
END_VAR
MesState := 0 ; 
IF MesOpened THEN		// If the cell seems opens and closed in the same time, we will consider it as opened. 
	
	MesState.0 := 1 ; 
MesDataExd.MesData.MesClosed := FALSE ; 
MesDataExd.MesData.MesOpened := TRUE ; 
ELSIF MesClosed THEN
	
	MesState.1 := 1 ; 
MesDataExd.MesData.MesClosed := TRUE ; 
MesDataExd.MesData.MesOpened := FALSE ; 
ELSE 
	MesState.0 := 1 ;		// if the cell seems neither opened and neither closed , we will consider it as opened. 
MesDataExd.MesData.MesClosed := FALSE ; 	
MesDataExd.MesData.MesOpened := TRUE ; 
END_IF
END_METHOD

END_FUNCTION_BLOCK

// ---- 01_Equipement_Library/Actuators/FB_CB_MVSwitch.TcPOU
FUNCTION_BLOCK FB_CB_MVSwitch EXTENDS FB_CB_Base
//////////////////
//  Motorized Circuit Breaker with telecommAND   Requires Open and Close impulsions.
//////////////////

VAR_INPUT PERSISTENT
	// Parameters of the Object (instance/model specific) 
	
END_VAR

VAR_INPUT
	// I/O Inputs              	
		
END_VAR

VAR
	//M_OPENCLOSE VARIABLES//

	
	//M_ALARMMANAGEMENT VARIABLES//
		
	//M_STATEMANAGER VARIABLES//
MesDataExd	       			 :  CB_Standard ; 
	// M_EXECUTE VARIABLES //
		
	// EMULATOR //

		
END_VAR

METHOD M_AlarmManagement
//////////////////
// Manages Contactor alarms and warnings
/////////////////

VAR 
	// Method local variables (reinitialized at each cycle) 
	FB_AlarmCodeManager			: FB_AlarmCodeManager ; 

	
END_VAR
VAR_INPUT
	
END_VAR
// Check if command and measures are matching after tempo
TON_NotClosedAndNotOpened(IN:=  NOT MesClosed AND NOT MesOpened , PT := ParamTimeOut_Alarm) ; 
TON_ClosedAndOpened(IN:= MesClosed AND MesOpened, PT := ParamTimeOut_Alarm) ; 
//RS_AlarmStopReclose(Set := MesTransfo_Fault, RESET1 := BlockWriteTemp[1] OR IN_CmdReset_L);

// ALARM CODE //
	FB_AlarmCodeManager(
		bAlarm1			:= FALSE, 									// 
		bAlarm2			:= TON_NotClosedAndNotOpened.Q,				// Incoherent State mesure (Not Opened and not Closed )
		bAlarm3 		:= TON_ClosedAndOpened.Q  , 				// Incoherent State mesure (Opened and Closed )	
		bAlarm4			:= FALSE, 									// 
		bAlarm5			:= FALSE, 									//
		bAlarm6			:= FALSE,                                   //
		bAlarm7			:= FALSE,                                   //
		bAlarm8			:= FALSE,                                   //
		bAlarm9			:= FALSE,                                   //
		bAlarm10		:= FALSE,                                   //
		bAlarm11		:= FALSE,                                   //
		bAlarm12		:= FALSE,                                   //
		bAlarm13		:= FALSE, 									//
		bAlarm14		:= FALSE, 									//
		bAlarm15		:= FALSE , 									// 
		wAlarmCode		=>MesDataExd.MesData.MesAlarmCode);

//WARNING CODE//
		FB_AlarmCodeManager(
		bAlarm1			:= FALSE , 									//
		bAlarm2			:= FALSE  , 		                        //
		bAlarm3 		:= FALSE,									//		
		bAlarm4			:= FALSE, 									//
		bAlarm5			:= FALSE,                                   //
		bAlarm6			:= FALSE,                                   //
		bAlarm7			:= FALSE,                                   //
		bAlarm8			:= FALSE,                                   //
		bAlarm9			:= FALSE,                                   //
		bAlarm10		:= FALSE,                                   //
		bAlarm11		:= FALSE,                                   //
		bAlarm12		:= FALSE,                                   //
		bAlarm13		:= FALSE,                                   //
		bAlarm14		:= FALSE,                                   //
		bAlarm15		:= FALSE,                                   //
		wAlarmCode 		=>MesDataExd.MesData.MesWarningCode);

// EVENT CODE //
	FB_AlarmCodeManager(
		bAlarm1			:= FALSE, 									// 
		bAlarm2			:= FALSE, 									// 
		bAlarm3			:= MesOpened, 								// Opened Position
		bAlarm4			:= MesClosed, 								// Closed Position
		bAlarm5			:= IN_CmdReset_L,                           // Reset Command
		bAlarm6			:= FALSE,                                   //
		bAlarm7			:= FALSE,                                   //
		bAlarm8			:= FALSE,                                   //
		bAlarm9			:= FALSE,                                   //
		bAlarm10		:= FALSE,                                   //
		bAlarm11		:= FALSE,                                   //
		bAlarm12		:= FALSE,                                   //
		bAlarm13		:= FALSE,                                   //
		bAlarm14		:= FALSE,                                   //
		bAlarm15		:= FALSE,                                   //
		wAlarmCode		=>MesDataExd.MesData.MesEventCode);
END_METHOD

METHOD M_Execute
VAR_INPUT
END_VAR
// PERMANENT CONDITIONS //	
MesDataExd.MesData.MesCP_Open					:= IN_CmdOpen AND NOT IN_CmdReset_L;
MesDataExd.MesData.MesCP_Close				:= NOT MesDataExd.MesData.MesClosed AND IN_CmdClose AND NOT MesDataExd.MesData.MesAlarmCode.0 AND NOT MesDataExd.MesData.MesCP_Open AND NOT IN_CmdReset_L ;


SUPER^.M_Execute();
END_METHOD

METHOD M_StateManager
//////////////////
// Manages Contactor State
/////////////////

VAR 
	// Method local variables (reinitialized at each cycle) 
	
END_VAR
MesState := 0 ; 
IF MesOpened THEN		// If the cell seems opens and closed in the same time, we will consider it as opened. 
	
	MesState.0 := 1 ; 
MesDataExd.MesData.MesClosed := FALSE ; 
MesDataExd.MesData.MesOpened := TRUE ; 
ELSIF MesClosed THEN
	
	MesState.1 := 1 ; 
MesDataExd.MesData.MesClosed := TRUE ; 
MesDataExd.MesData.MesOpened := FALSE ; 
ELSE 
	MesState.0 := 1 ;		// if the cell seems neither opened and neither closed , we will consider it as opened. 
MesDataExd.MesData.MesClosed := FALSE ; 	
MesDataExd.MesData.MesOpened := TRUE ; 
END_IF
END_METHOD

END_FUNCTION_BLOCK

// ---- 01_Equipement_Library/Actuators/FB_CB_MainMVCB.TcPOU
FUNCTION_BLOCK FB_CB_MainMVCB EXTENDS FB_CB_Base
//////////////////
//  Motorized Circuit Breaker with telecommAND  Requires Open and Close impulsions.
//////////////////

VAR_INPUT PERSISTENT
	// Parameters of the Object (instance/model specific) 
	ParamTP_Impulsion		    : TIME 		:= T#2S;	(* (s) Config : Tempo for the start or stop command impulsion*)
	ParamComutNc			    : BOOL;					(* (NA) Local selector in normally closed. NC >> True = Selector in local *)
	ParamSectLigne			    : BYTE      :=1;		(* (NA) Monitoring du sectionneur de ligne de la MainMVCB . 0 = TRUE := Monitoré . 1 = TRUE Close is connected*)
	ParamUvCoil					: BOOL;					(* (NA) if the open and close order are linked to a undervoltage coil (Bobine à manque, Bobine Mn), this should be True*)
END_VAR

VAR_OUTPUT
	//Child objects
	OUT_CmdOpen_IO	           : BOOL ; 	          // (NA) Physical I/O Open Command IO
	OUT_CmdClose_IO			   : BOOL ; 	          // (NA) Physical I/O Close Command IO
	OUT_CmdMaintainClose_IO		: BOOL;					// (NA) Physical I/O close for the UV coil.
END_VAR

VAR_INPUT
	A1_Sect				        : FB_CB_MVSwitch;

// I/O Inputs              
	IN_MesAlarmPwr_IO		    : BOOL ;	          // (NA)[P,H,B] Remote control Power supply Error  IO  	
	IN_MesTripped_IO		  	: BOOL ; 	          // (NA) Tripped position of the CB Must Ack To switch in again
	IN_MesComutLocal_IO			: BOOL := TRUE ; 	  // (NA) True if cell is in local position  
	IN_MesEarth_IO 			    : BOOL ; 	


	MesDataExd			        :  CB_MainMVCB_Sch ; 
		
END_VAR

VAR
	//M_OPENCLOSE VARIABLES//	
		ParamTP_Open	 			: TP ;				(* (NA) Temporisation for Open pulse Command*)
		ParamTP_Close 				: TP ;				(* (NA) Temporisation for Close pulse Command	*)
		RS_MaintainClose					: RS ;				(* (NA) RS to manage UV Coil*)
	//M_ALARMMANAGEMENT VARIABLES//
	
//M_STATEMANAGER VARIABLES//
	
END_VAR

METHOD M_AlarmManagement
//////////////////
// Manages Contactor alarms and warnings
/////////////////

VAR 
	// Method local variables (reinitialized at each cycle) 
	FB_AlarmCodeManager			: FB_AlarmCodeManager ; 
	
	CmdOpenCloseIO				: BOOL; 				//Check IN/OUT_CMDOpenClose
	bSectLigne					: BOOL;
END_VAR
// Check if command and measures are matching after tempo
FB_CheckCommand	(T:= ParamTimeOut_Close, bCmd:=OUT_CmdClose_IO , bMes := MesDataExd.MesData.MesClosed , bImpulsion := FALSE , bReset := CmdClearFault_G OR OUT_CmdClose_IO) ; 
FB_CheckCommand2(T:= ParamTimeOut_Open , bCmd:= OUT_CmdOpen_IO , bMes :=NOT MesDataExd.MesData.MesClosed , bImpulsion := FALSE , bReset := CmdClearFault_G OR OUT_CmdOpen_IO) ; 

TON_NotClosedAndNotOpened(IN:=  NOT MesClosed AND NOT MesOpened , PT := ParamTimeOut_Alarm) ; 
TON_ClosedAndOpened(IN:=MesClosed AND MesOpened, PT := ParamTimeOut_Alarm) ; 


// ALARM CODE //
	FB_AlarmCodeManager(
		bAlarm1			:= MesDataExd.MesTripped,						// Cb is tripped
		bAlarm2			:= TON_NotClosedAndNotOpened.Q,					// Incoherent State mesure (Not Opened and not Closed)
		bAlarm3 		:= TON_ClosedAndOpened.Q,	 					// Incoherent State mesure (Opened and Closed)	
		bAlarm4			:= FB_CheckCommAND.bWarning, 					// Close command failed
		bAlarm5			:= FB_CheckCommand2.bWarning,	 				// Open Command failed
		bAlarm6			:= FALSE,                                   	//
		bAlarm7			:= FALSE,                                   	//
		bAlarm8			:= FALSE,                                   	//
		bAlarm9			:= FALSE,                                   	//
		bAlarm10		:= FALSE,                                   	//
		bAlarm11		:= FALSE,                                   	//
		bAlarm12		:= FALSE,                                   	//
		bAlarm13		:= FALSE,                                   	//
		bAlarm14		:= FALSE,                                   	//
		bAlarm15		:= FALSE , 										//
		wAlarmCode		=>MesDataExd.MesData.MesAlarmCode);

	bSectLigne := SEL(ParamSectLigne.0 ,FALSE , NOT A1_Sect.MesDataExd.MesData.MesClosed);
//WARNING CODE//
		FB_AlarmCodeManager(
		bAlarm1			:= FALSE,										//
		bAlarm2			:= FALSE,										//
		bAlarm3 		:= FALSE,										// 
		bAlarm4			:= MesDataExd.MesAlarmPwr, 						// Power Supply Fault
		bAlarm5			:= MesDataExd.MesComutLocal, 					// Commutator in local mode 
		bAlarm6			:= MesDataExd.MesEarth, 						// The cell is connected to earth (earthing)
		bAlarm7			:= bSectLigne,									// Line connector is opened (sectionneur)
		bAlarm8			:= FALSE, 										//
		bAlarm9			:= FALSE,                                       //
		bAlarm10		:= FALSE,                                       //
		bAlarm11		:= FALSE,                                       //
		bAlarm12		:= FALSE,                                       //
		bAlarm13		:= FALSE,                                       //
		bAlarm14		:= FALSE,                                       //
		bAlarm15		:= FALSE, 										//
		wAlarmCode 		=>MesDataExd.MesData.MesWarningCode);

// EVENT CODE //
	FB_AlarmCodeManager(
		bAlarm1			:= OUT_CmdOpen_IO, 								// Open Command
		bAlarm2			:= OUT_CmdClose_IO, 							// Close Comamnd
		bAlarm3			:= MesOpened, 									// Opened Position
		bAlarm4			:= MesClosed, 									// Closed Position
		bAlarm5			:= IN_CmdReset_L, 								// Reset command
		bAlarm6			:= FALSE, 										//
		bAlarm7			:= FALSE,                   					//
		bAlarm8			:= FALSE,                   					//
		bAlarm9			:= FALSE,                   					//
		bAlarm10		:= FALSE,                   					//
		bAlarm11		:= FALSE,                   					//
		bAlarm12		:= FALSE,                   					//
		bAlarm13		:= FALSE, 										//
		bAlarm14		:= FALSE,                   					//
		bAlarm15		:= FALSE,                   					//
		wAlarmCode		=>MesDataExd.MesData.MesEventCode);                                               
	                                                
	// UPDATE STRUCTURE
	
	IF ParamComutNc THEN
	MesDataExd.MesComutLocal	:= NOT IN_MesComutLocal_IO ; 
	ELSE
	MesDataExd.MesComutLocal	:= IN_MesComutLocal_IO ; 
	END_IF
	
MesDataExd.MesAlarmPwr		    := IN_MesAlarmPwr_IO ; 
MesDataExd.MesTripped			:= IN_MesTripped_IO ; 
MesDataExd.OUT_CmdClose		    := OUT_CmdClose_IO ; 
MesDataExd.OUT_CmdOpen		    := OUT_CmdOpen_IO ; 
MesDataExd.MesEarth			    := IN_MesEarth_IO ; 
MesDataExd.MesOpened_Sect	    := SEL(ParamSectLigne.0, FALSE, A1_Sect.MesDataExd.MesData.MesOpened) ;
END_METHOD

METHOD M_Execute
VAR_INPUT
END_VAR

VAR

END_VAR
//MainMVCB avec etat de sectionneur de ligne
IF ParamSectLigne.0 THEN 
	A1_Sect.ParamNbFdbck := 1;
	A1_Sect.ParamNC := ParamSectLigne.1;
	A1_Sect.ParamClosedInput_Connected := TRUE ; 
	A1_Sect.M_Execute();
END_IF

// PERMANENT CONDITIONS //	
MesDataExd.MesData.MesCP_Open					:= IN_CmdOpen AND NOT IN_CmdReset_L;
MesDataExd.MesData.MesCP_Close				:= NOT MesDataExd.MesData.MesClosed AND IN_CmdClose AND NOT MesDataExd.MesData.MesAlarmCode.0 AND NOT MesDataExd.MesData.MesCP_Open AND NOT IN_CmdReset_L ;


SUPER^.M_Execute();
END_METHOD

METHOD M_OpenClose
//////////////////
// Manages Opening and Closing of the contactor
//////////////////

VAR 
	// Method local variables (reinitialized at each cycle) 

	
END_VAR
//AJOUT EXEPTION MAIN CIRCUIT BREAKER 
IF ParamSectLigne.0 THEN
	MesDataExd.MesData.MesCP_Close := MesDataExd.MesData.MesCP_Close AND NOT MesDataExd.MesOpened_Sect; // A1_Sect.IN_MesClosed_IO; //Check
END_IF
(*

Il peut y avoir 3 bobines :
 Bobine d'ouverture = on envoie un créneau pour fermer la cellule
 Bobine de fermeture = on envoie un créneau pour ouvrir la cellule
 Bobine à manque = si pas alimentée, la cellule ne peut pas rester fermée ni se fermer.
 Dans certaines cellules, il n'y a pas de bobine d'ouverture : il faut enlever l'alimentation de la bobine à manque pour que la cellule s'ouvre. 

*)

// ATTENTION : CODE NON TESTE ENCORE.
IF ParamUvCoil THEN
	RS_MaintainClose(set := MesDataExd.MesData.MesCP_Close OR NOT MesDataExd.MesData.MesCP_Open, RESET1 := MesDataExd.MesData.MesCP_Open);
	// je pourrais mettre que le Not CP_Open : il me permet d'être sûr que la bobine à manque est désactivée que quelques secondes
	OUT_CmdMaintainClose_IO := RS_MaintainClose.Q1;
END_IF


// Open Command
	ParamTP_Open(IN:= MesDataExd.MesData.MesCP_Open , PT:=ParamTP_Impulsion) ;
	OUT_CmdOpen_IO	 := ParamTP_Open.Q ;	// Impulsion that goes back to zero as soon as the state of the TP goes down. 

// Close Command
	ParamTP_Close(IN:= MesDataExd.MesData.MesCP_Close , PT:=ParamTP_Impulsion) ;
	OUT_CmdClose_IO	 := ParamTP_Close.Q ;   // Impulsion that goes back to zero as soon as the state of the TP goes down.
END_METHOD

METHOD M_StateManager
//////////////////
// Manages Contactor State
/////////////////

VAR 
	// Method local variables (reinitialized at each cycle) 
	
END_VAR
MesState := 0 ; 
IF MesOpened THEN		// If the cell seems opens and closed in the same time, we will consider it as opened. 
	
	MesState.0 := 1 ; 
MesDataExd.MesData.MesClosed := FALSE ; 
MesDataExd.MesData.MesOpened := TRUE ; 
ELSIF MesClosed THEN
	
	MesState.1 := 1 ; 
MesDataExd.MesData.MesClosed := TRUE ; 
MesDataExd.MesData.MesOpened := FALSE ; 
ELSE 
	MesState.0 := 1 ;		// if the cell seems neither opened and neither closed , we will consider it as opened. 
MesDataExd.MesData.MesClosed := FALSE ; 	
MesDataExd.MesData.MesOpened := TRUE ; 
END_IF
END_METHOD

END_FUNCTION_BLOCK

// ---- 01_Equipement_Library/Actuators/FB_CB_MeasureMVCB.TcPOU
FUNCTION_BLOCK FB_CB_MeasureMVCB EXTENDS FB_CB_Base
//////////////////
//  Motorized Circuit Breaker with telecommAND  Requires Open and Close impulsions.
//////////////////

VAR_INPUT PERSISTENT
	// Parameters of the Object (instance/model specific) 
	ParamTP_Impulsion	   : TIME := T#2S;			(* (s) 	 Config : Tempo for the start or stop command impulsion*)
	ParamFuseNC		       : BOOL;					(* (NA)	 False  : TRUE = Closed , True : TRUE = opened	*)
END_VAR

VAR_OUTPUT
	//Child objects
	
END_VAR

VAR_INPUT
	// I/O Inputs              
	IN_MesFuse_IO			: BOOL;
	IN_MesEarth_IO			: BOOL; 
	
END_VAR

VAR
	//M_OPENCLOSE VARIABLES//	
		RsFuse				: RS ;
		
	//M_ALARMMANAGEMENT VARIABLES//
	MesDataExd	: CB_MeasureMVCB_Sch ;
 
	//M_STATEMANAGER VARIABLES//
	
	// M_EXECUTE VARIABLES //
	
END_VAR

METHOD M_AlarmManagement
//////////////////
// Manages Contactor alarms and warnings
/////////////////

VAR 
	// Method local variables (reinitialized at each cycle) 
	FB_AlarmCodeManager			: FB_AlarmCodeManager ; 

	
END_VAR
// Check if command and measures are matching after tempo

TON_NotClosedAndNotOpened(IN:=  NOT MesClosed AND NOT MesOpened , PT := ParamTimeOut_Alarm) ; 
TON_ClosedAndOpened(IN:=MesClosed AND MesOpened, PT := ParamTimeOut_Alarm) ; 

RsFuse(Set:= MesDataExd.MesFuseBurned ,Reset1:=GVL_CFG.CmdClearFault_G OR IN_CmdReset_L);



// ALARM CODE //
	FB_AlarmCodeManager(
		bAlarm1			:= FALSE,										//
		bAlarm2			:= TON_NotClosedAndNotOpened.Q,					// Incoherent State mesure (Not Opened and not Closed 
		bAlarm3 		:= TON_ClosedAndOpened.Q   , 					// Incoherent State mesure (Opened and Closed )	
		bAlarm4			:= RsFuse.Q1,									// Fuse burned
		bAlarm5			:= FALSE, 										//  
		bAlarm6			:= FALSE, 										//
		bAlarm7			:= FALSE,                                       //
		bAlarm8			:= FALSE,                                       //
		bAlarm9			:= FALSE,                                       //
		bAlarm10		:= FALSE,                                       //
		bAlarm11		:= FALSE,                                       //
		bAlarm12		:= FALSE,                                       //
		bAlarm13		:= FALSE, 										//
		bAlarm14		:= FALSE, 										//
		bAlarm15		:= FALSE , 										// 
		wAlarmCode		=>MesDataExd.MesData.MesAlarmCode);

//WARNING CODE//
		FB_AlarmCodeManager(
		bAlarm1			:= FALSE , 										// 
		bAlarm2			:= FALSE  , 									// 
		bAlarm3 		:= FALSE,										// 
		bAlarm4			:= FALSE, 										// 
		bAlarm5			:= FALSE, 										//
		bAlarm6			:= MesDataExd.MesEarth, 						// Earthing
		bAlarm7			:= FALSE, 										//
		bAlarm8			:= FALSE,                                       //
		bAlarm9			:= FALSE,                                       //
		bAlarm10		:= FALSE,                                       //
		bAlarm11		:= FALSE,                                       //
		bAlarm12		:= FALSE,                                       //
		bAlarm13		:= FALSE,                                       //
		bAlarm14		:= FALSE,                                       //
		bAlarm15		:= FALSE, 										//
		wAlarmCode 		=>MesDataExd.MesData.MesWarningCode);

// EVENT CODE //
	FB_AlarmCodeManager(
		bAlarm1			:= FALSE, 										// 
		bAlarm2			:= FALSE, 										// 
		bAlarm3			:= MesOpened, 									// Opened Position
		bAlarm4			:= MesClosed, 									// Closed Position
		bAlarm5			:= IN_CmdReset_L, 								// Reset Command
		bAlarm6			:= FALSE, 										//
		bAlarm7			:= FALSE,                                       //
		bAlarm8			:= FALSE,                                       //
		bAlarm9			:= FALSE,                                       //
		bAlarm10		:= FALSE,                                       //
		bAlarm11		:= FALSE,                                       //
		bAlarm12		:= FALSE,                                       //
		bAlarm13		:= FALSE,                                       //
		bAlarm14		:= FALSE, 										//
		bAlarm15		:= FALSE, 										//
		wAlarmCode		=>MesDataExd.MesData.MesEventCode);
		
	// UPDATE STRUCTURE


		
	IF NOT ParamFuseNC THEN 
	MesDataExd.MesFuseBurned := NOT IN_MesFuse_IO;
	ELSE
	MesDataExd.MesFuseBurned := IN_MesFuse_IO;
	END_IF
	
MesDataExd.MesEarth	:= IN_MesEarth_IO ;
END_METHOD

METHOD M_Execute
VAR_INPUT
END_VAR

// PERMANENT CONDITIONS //	
MesDataExd.MesData.MesCP_Open					:= IN_CmdOpen AND NOT IN_CmdReset_L;
MesDataExd.MesData.MesCP_Close				:= NOT MesDataExd.MesData.MesClosed AND IN_CmdClose AND NOT MesDataExd.MesData.MesAlarmCode.0 AND NOT MesDataExd.MesData.MesCP_Open AND NOT IN_CmdReset_L ;


SUPER^.M_Execute();
END_METHOD

METHOD M_OpenClose
//////////////////
// Manages Opening and Closing of the contactor
//////////////////

VAR 
	// Method local variables (reinitialized at each cycle) 

	
END_VAR
END_METHOD

METHOD M_StateManager
//////////////////
// Manages Contactor State
/////////////////

VAR 
	// Method local variables (reinitialized at each cycle) 
	
END_VAR
MesState := 0 ; 
IF MesOpened THEN		// If the cell seems opens and closed in the same time, we will consider it as opened. 
	
	MesState.0 := 1 ; 
MesDataExd.MesData.MesClosed := FALSE ; 
MesDataExd.MesData.MesOpened := TRUE ; 
ELSIF MesClosed THEN
	
	MesState.1 := 1 ; 
MesDataExd.MesData.MesClosed := TRUE ; 
MesDataExd.MesData.MesOpened := FALSE ; 
ELSE 
	MesState.0 := 1 ;		// if the cell seems neither opened and neither closed , we will consider it as opened. 
MesDataExd.MesData.MesClosed := FALSE ; 	
MesDataExd.MesData.MesOpened := TRUE ; 
END_IF
END_METHOD

END_FUNCTION_BLOCK

// ---- 01_Equipement_Library/Actuators/FB_CB_AuxMVCB.TcPOU
FUNCTION_BLOCK FB_CB_AuxMVCB EXTENDS FB_CB_Base
//////////////////
//  Motorized Circuit Breaker with telecommAND   Requires Open and Close impulsions.
//////////////////

VAR_INPUT PERSISTENT
	// Parameters of the Object (instance/model specific) 
	ParamTP_Impulsion	   : TIME := T#2S;			(* (s)  Config : Tempo for the start or stop command impulsion*)
	ParamFuseNC		       : BOOL;					(* (NA) False: TRUE = Closed , True : TRUE = opened	*)
END_VAR

VAR_OUTPUT
	//Child objects
	
END_VAR

VAR_INPUT
	// I/O Inputs              
	IN_MesFuse_IO			: BOOL;
	IN_MesEarth_IO			: BOOL; 
	
END_VAR

VAR
	//M_OPENCLOSE VARIABLES//	
		RsFuse				:RS;
		
	//M_ALARMMANAGEMENT VARIABLES//
	MesDataExd	: CB_AuxMVCB_Sch;
 
	//M_STATEMANAGER VARIABLES//
	
	// M_EXECUTE VARIABLES //
		
 
END_VAR

METHOD M_AlarmManagement
//////////////////
// Manages Contactor alarms and warnings
/////////////////

VAR 
	// Method local variables (reinitialized at each cycle) 
	FB_AlarmCodeManager			: FB_AlarmCodeManager ; 	
END_VAR
// Check if command and measures are matching after tempo

TON_NotClosedAndNotOpened(IN:=  NOT MesClosed AND NOT MesOpened , PT := ParamTimeOut_Alarm) ; 
TON_ClosedAndOpened(IN:=MesClosed AND MesOpened, PT := ParamTimeOut_Alarm) ; 

RsFuse(Set:= MesDataExd.MesFuseBurned ,Reset1:=GVL_CFG.CmdClearFault_G OR IN_CmdReset_L);

// ALARM CODE //
	FB_AlarmCodeManager(
		bAlarm1			:= FALSE,										//
		bAlarm2			:= TON_NotClosedAndNotOpened.Q,					// Incoherent state mesure (neither open nor closed) 
		bAlarm3 		:= TON_ClosedAndOpened.Q, 						// Incoherent state mesure (Open and closed)	
		bAlarm4			:= RsFuse.Q1,									// Fuse is burned
		bAlarm5			:= FALSE, 										//  
		bAlarm6			:= FALSE, 										//
		bAlarm7			:= FALSE,                                       //
		bAlarm8			:= FALSE,                                       //
		bAlarm9			:= FALSE,                                       //
		bAlarm10		:= FALSE,                                       //
		bAlarm11		:= FALSE,                                       //
		bAlarm12		:= FALSE,                                       //
		bAlarm13		:= FALSE, 										//
		bAlarm14		:= FALSE, 										//
		bAlarm15		:= FALSE , 										// 
		wAlarmCode		=>MesDataExd.MesData.MesAlarmCode);

//WARNING CODE//
		FB_AlarmCodeManager(
		bAlarm1			:= FALSE, 										// 
		bAlarm2			:= FALSE,	 									// 
		bAlarm3 		:= FALSE,										// 
		bAlarm4			:= FALSE, 										// 
		bAlarm5			:= FALSE, 										//
		bAlarm6			:= MesDataExd.MesEarth, 						// Earthing mode
		bAlarm7			:= FALSE, 										//
		bAlarm8			:= FALSE,                                       //
		bAlarm9			:= FALSE,                                       //
		bAlarm10		:= FALSE,                                       //
		bAlarm11		:= FALSE,                                       //
		bAlarm12		:= FALSE,                                       //
		bAlarm13		:= FALSE,                                       //
		bAlarm14		:= FALSE,                                       //
		bAlarm15		:= FALSE, 										//
		wAlarmCode 		=>MesDataExd.MesData.MesWarningCode);

// EVENT CODE //
	FB_AlarmCodeManager(
		bAlarm1			:= FALSE, 										// 
		bAlarm2			:= FALSE, 										// 
		bAlarm3			:= MesOpened, 									// Open position
		bAlarm4			:= MesClosed, 									// Closed position
		bAlarm5			:= IN_CmdReset_L, 								// Reset Command
		bAlarm6			:= FALSE, 										//
		bAlarm7			:= FALSE,                                       //
		bAlarm8			:= FALSE,                                       //
		bAlarm9			:= FALSE,                                       //
		bAlarm10		:= FALSE,                                       //
		bAlarm11		:= FALSE,                                       //
		bAlarm12		:= FALSE,                                       //
		bAlarm13		:= FALSE,                                       //
		bAlarm14		:= FALSE, 										//
		bAlarm15		:= FALSE, 										//
		wAlarmCode		=>MesDataExd.MesData.MesEventCode);
		
	// UPDATE STRUCTURE


	IF NOT ParamFuseNC THEN 
	MesDataExd.MesFuseBurned := NOT IN_MesFuse_IO;
	ELSE
	MesDataExd.MesFuseBurned := IN_MesFuse_IO;
	END_IF
MesDataExd.MesEarth	:= IN_MesEarth_IO ;
END_METHOD

METHOD M_Execute
VAR_INPUT
END_VAR
// PERMANENT CONDITIONS //	
MesDataExd.MesData.MesCP_Open					:= IN_CmdOpen AND NOT IN_CmdReset_L;
MesDataExd.MesData.MesCP_Close				:= NOT MesDataExd.MesData.MesClosed AND IN_CmdClose AND NOT MesDataExd.MesData.MesAlarmCode.0 AND NOT MesDataExd.MesData.MesCP_Open AND NOT IN_CmdReset_L ;


SUPER^.M_Execute();
END_METHOD

METHOD M_OpenClose
//////////////////
// Manages Opening and Closing of the contactor
//////////////////

VAR 
	// Method local variables (reinitialized at each cycle) 

	
END_VAR
END_METHOD

METHOD M_StateManager
//////////////////
// Manages Contactor State
/////////////////

VAR 
	// Method local variables (reinitialized at each cycle) 
	
END_VAR
MesState := 0 ; 
IF MesOpened THEN		// If the cell seems opens and closed in the same time, we will consider it as opened. 
	
	MesState.0 := 1 ; 
MesDataExd.MesData.MesClosed := FALSE ; 
MesDataExd.MesData.MesOpened := TRUE ; 
ELSIF MesClosed THEN
	
	MesState.1 := 1 ; 
MesDataExd.MesData.MesClosed := TRUE ; 
MesDataExd.MesData.MesOpened := FALSE ; 
ELSE 
	MesState.0 := 1 ;		// if the cell seems neither opened and neither closed , we will consider it as opened. 
MesDataExd.MesData.MesClosed := FALSE ; 	
MesDataExd.MesData.MesOpened := TRUE ; 
END_IF
END_METHOD

END_FUNCTION_BLOCK

// ---- 01_Equipement_Library/Actuators/FB_CB_FeederMVCB.TcPOU
FUNCTION_BLOCK FB_CB_FeederMVCB EXTENDS FB_CB_Base
//////////////////
//  Motorized Circuit Breaker with telecommAND   Requires Open and Close impulsions.
//////////////////

VAR_INPUT PERSISTENT
	// Parameters of the Object (instance/model specific) 
	ParamTP_Impulsion		    : TIME 		:= T#2S;	(* (s) Config : Tempo for the start or stop command impulsion*)
	ParamComutNc			    : BOOL;					(* (NA) Local selector in normally closed. NC >> True = Selector in local. *)
	ParamSectLigne			    : BYTE      :=1;		(* (NA) Monitoring du sectionneur de ligne de la MainMVCB.0 = TRUE := Monitoré .1 = TRUE Close is connected*)

END_VAR
VAR_INPUT
	A1_Sect				       : FB_CB_MVSwitch;

// I/O Inputs              
	IN_MesAlarmPwr_IO		   : BOOL ;	              // (NA)[P,H,B] Remote control Power supply Error IO  	
	IN_MesTripped_IO		   : BOOL ; 	          // Tripped position of the CB Must Ack To switch in again
	IN_MesComutLocal_IO		   : BOOL ;	 	 		 // True if cell is in local position 
	IN_MesEarth_IO 			   : BOOL ; 	
		
END_VAR

VAR_OUTPUT
	//Child objects
	OUT_CmdOpen_IO	           : BOOL ; 	          // (NA) Physical I/O Open Command IO
	OUT_CmdClose_IO			   : BOOL ; 	          // (NA) Physical I/O Close Command IO
	
END_VAR


VAR
	//M_OPENCLOSE VARIABLES//
	MesDataExd					: CB_FeederMVCB_Sch ; 
	//M_OPENCLOSE VARIABLES//	
	ParamTP_Open	 			: TP ;				(* (NA) Temporisation for Open pulse Command*)
	ParamTP_Close 				: TP ;				(* (NA) Temporisation for Close pulse Command	*)
		
END_VAR

METHOD M_AlarmManagement
//////////////////
// Manages Contactor alarms and warnings
/////////////////

VAR 
	// Method local variables (reinitialized at each cycle) 
	FB_AlarmCodeManager			: FB_AlarmCodeManager ; 
	bSectLigne					: BOOL;
END_VAR
VAR_INPUT
	
END_VAR
// Check if command and measures are matching after tempo
FB_CheckCommand	(T:= ParamTimeOut_Close, bCmd:=OUT_CmdClose_IO , bMes := MesDataExd.MesData.MesClosed , bImpulsion := FALSE , bReset := CmdClearFault_G OR OUT_CmdClose_IO) ; 
FB_CheckCommand2(T:= ParamTimeOut_Open , bCmd:= OUT_CmdOpen_IO , bMes :=NOT MesDataExd.MesData.MesClosed , bImpulsion := FALSE , bReset := CmdClearFault_G OR OUT_CmdOpen_IO) ; 

TON_NotClosedAndNotOpened(IN:=  NOT MesClosed AND NOT MesOpened , PT := ParamTimeOut_Alarm) ; 
TON_ClosedAndOpened(IN:=MesClosed AND MesOpened, PT := ParamTimeOut_Alarm) ; 

// ALARM CODE //
	FB_AlarmCodeManager(
		bAlarm1			:= MesDataExd.MesTripped,						// CB is tripped
		bAlarm2			:= TON_NotClosedAndNotOpened.Q,					// Incoherent State mesure (Not Opened and not Closed)
		bAlarm3 		:= TON_ClosedAndOpened.Q   , 					// Incoherent State mesure (Opened and Closed)	
		bAlarm4			:= FB_CheckCommAND.bWarning , 					// Close command failed
		bAlarm5			:= FB_CheckCommand2.bWarning  , 				// Open Command failed
		bAlarm6			:= FALSE,                                   	//
		bAlarm7			:= FALSE,                                   	//
		bAlarm8			:= FALSE,                                   	//
		bAlarm9			:= FALSE,                                   	//
		bAlarm10		:= FALSE,                                   	//
		bAlarm11		:= FALSE,                                   	//
		bAlarm12		:= FALSE,                                   	//
		bAlarm13		:= FALSE,                                   	//
		bAlarm14		:= FALSE,                                   	//
		bAlarm15		:= FALSE , 										//
		wAlarmCode		=>MesDataExd.MesData.MesAlarmCode);

		
	bSectLigne := SEL(ParamSectLigne.0 ,FALSE , NOT A1_Sect.MesDataExd.MesData.MesClosed);
//WARNING CODE//
		FB_AlarmCodeManager(
		bAlarm1			:= FALSE,										//
		bAlarm2			:= FALSE,										//
		bAlarm3 		:= FALSE,										// 
		bAlarm4			:= MesDataExd.MesAlarmPwr, 						// Power supply fault
		bAlarm5			:= MesDataExd.MesComutLocal, 					// Comutator in LOCAL mode
		bAlarm6			:= MesDataExd.MesEarth, 						// Earthing is done 
		bAlarm7			:= bSectLigne,	// Line sectionnor is opened
		bAlarm8			:= FALSE, 										//
		bAlarm9			:= FALSE,                                       //
		bAlarm10		:= FALSE,                                       //
		bAlarm11		:= FALSE,                                       //
		bAlarm12		:= FALSE,                                       //
		bAlarm13		:= FALSE,                                       //
		bAlarm14		:= FALSE,                                       //
		bAlarm15		:= FALSE, 										//
		wAlarmCode 		=>MesDataExd.MesData.MesWarningCode);

// EVENT CODE //
	FB_AlarmCodeManager(
		bAlarm1			:= OUT_CmdOpen_IO, 								// Open Command
		bAlarm2			:= OUT_CmdClose_IO, 							// Close Comamnd
		bAlarm3			:= MesOpened, 									// Opened Position
		bAlarm4			:= MesClosed, 									// Closed Position
		bAlarm5			:= IN_CmdReset_L, 								// Reset command
		bAlarm6			:= FALSE, 										//
		bAlarm7			:= FALSE,                   					//
		bAlarm8			:= FALSE,                   					//
		bAlarm9			:= FALSE,                   					//
		bAlarm10		:= FALSE,                   					//
		bAlarm11		:= FALSE,                   					//
		bAlarm12		:= FALSE,                   					//
		bAlarm13		:= FALSE, 										//
		bAlarm14		:= FALSE,                   					//
		bAlarm15		:= FALSE,                   					//
		wAlarmCode		=>MesDataExd.MesData.MesEventCode);   
                                           
	// UPDATE STRUCTURE	
	IF ParamComutNc THEN
	MesDataExd.MesComutLocal	:= NOT IN_MesComutLocal_IO ; 
	ELSE
	MesDataExd.MesComutLocal	:= IN_MesComutLocal_IO ; 
	END_IF
	
MesDataExd.MesAlarmPwr		    := IN_MesAlarmPwr_IO ; 
MesDataExd.MesTripped			:= IN_MesTripped_IO ; 
MesDataExd.OUT_CmdClose		    := OUT_CmdClose_IO ; 
MesDataExd.OUT_CmdOpen		    := OUT_CmdOpen_IO ; 
MesDataExd.MesEarth			    := IN_MesEarth_IO ; 
MesDataExd.MesOpened_Sect	        := SEL(ParamSectLigne.0 , FALSE  , NOT A1_Sect.MesDataExd.MesData.MesClosed ) ; 
	
	//MesDataExd	    := MesDataExd.MesData.;
END_METHOD

METHOD M_Execute
VAR_INPUT
END_VAR

VAR

END_VAR
//MainMVCB avec etat de sectionneur de ligne
IF ParamSectLigne.0 THEN 
	A1_Sect.ParamNbFdbck := 1;
	A1_Sect.ParamNC := ParamSectLigne.1;
	A1_Sect.ParamClosedInput_Connected := TRUE ; 
	A1_Sect.M_Execute();
END_IF

// PERMANENT CONDITIONS //	
MesDataExd.MesData.MesCP_Open					:= IN_CmdOpen AND NOT IN_CmdReset_L;
MesDataExd.MesData.MesCP_Close				:= NOT MesDataExd.MesData.MesClosed AND IN_CmdClose AND NOT MesDataExd.MesData.MesAlarmCode.0 AND NOT MesDataExd.MesData.MesCP_Open AND NOT IN_CmdReset_L ;


SUPER^.M_Execute();
END_METHOD

METHOD M_OpenClose
//////////////////
// Manages Opening and Closing of the contactor
//////////////////

VAR 
	// Method local variables (reinitialized at each cycle) 

	
END_VAR
//AJOUT EXEPTION MAIN CIRCUIT BREAKER 
IF ParamSectLigne.0 THEN
MesDataExd.MesData.MesCP_Close := MesDataExd.MesData.MesCP_Close AND A1_Sect.IN_MesClosed_IO; //Check
END_IF

// Open Command
ParamTP_Open(IN:= MesDataExd.MesData.MesCP_Open , PT:=ParamTP_Impulsion) ;
OUT_CmdOpen_IO	 := ParamTP_Open.Q ;                               			 // Impulsion that goes back to zero as soon as the state of the TP goes down. 

// Close Command
ParamTP_Close(IN:= MesDataExd.MesData.MesCP_Close , PT:=ParamTP_Impulsion) ;
OUT_CmdClose_IO	 := ParamTP_Close.Q ;                          			 // Impulsion that goes back to zero as soon as the state of the TP goes down.
END_METHOD

METHOD M_StateManager
//////////////////
// Manages Contactor State
/////////////////

VAR 
	// Method local variables (reinitialized at each cycle) 
	
END_VAR
MesState := 0 ; 
IF MesOpened THEN		// If the cell seems opens and closed in the same time, we will consider it as opened. 
	
	MesState.0 := 1 ; 
MesDataExd.MesData.MesClosed := FALSE ; 
MesDataExd.MesData.MesOpened := TRUE ; 
ELSIF MesClosed THEN
	
	MesState.1 := 1 ; 
MesDataExd.MesData.MesClosed := TRUE ; 
MesDataExd.MesData.MesOpened := FALSE ; 
ELSE 
	MesState.0 := 1 ;		// if the cell seems neither opened and neither closed , we will consider it as opened. 
MesDataExd.MesData.MesClosed := FALSE ; 	
MesDataExd.MesData.MesOpened := TRUE ; 
END_IF
END_METHOD

END_FUNCTION_BLOCK

// ---- 01_Equipement_Library/Datalogger/FB_Datalogger_Base.TcPOU
FUNCTION_BLOCK FB_Datalogger_Base

VAR_INPUT PERSISTENT
	ParamTcpPort				: UINT	:=	502;		 (* (NA) Modbus TCP port*)
	ParamIPAddress				: STRING;				 (* (NA) Config: IP Adress *)
	ParamUnitID					: BYTE;					 (* (NA) Modbus Unit ID *)
	ParamClockRead 				: TIME 	:= TIME#2S; 	 (* (Time) Read Modbus frequency  	*)
	
	bInit						: BOOL  := TRUE; 		 // (NA) Initialisation 
END_VAR

VAR_INPUT           	
	IN_CmdToggleRead			: BOOL;
	IN_CmdToggleWrite			: BOOL;
	IN_CmdReset_L				: BOOL;
END_VAR             	
      	
VAR                 	
//INPUT
	ClockRead					: BOOL;							// (NA) Modbus reading Clock
    TP1							: TP ; 							// (NA) Tempo to define Modbus Reading Frequency 
	
	Trig_Cmd_Read				: R_Trig;
	Trig_Cmd_Write              : R_Trig;

	
		MesCP_Read					: BOOL := TRUE;	(* Read function enable *)
		MesCP_Write					: BOOL := TRUE;	(* Write function enable *)	
	
	
//  MesDataExd.MesData.                    : Datalogger;
END_VAR

VAR PERSISTENT

END_VAR

METHOD M_AlarmManagement
//////////////////
// Generates object alarms and manages resets. 
//////////////////

VAR 
	// Method local variables (reinitialized at each cycle) 
	FB_AlarmCodeManager		: FB_AlarmCodeManager ;  
END_VAR
END_METHOD

METHOD M_CP

VAR 
	// Method local variables (reinitialized at each cycle) 
	
END_VAR


Trig_Cmd_Write(CLK:=  IN_CmdToggleWrite);
	
Trig_Cmd_Read(CLK:=IN_CmdToggleRead);


IF Trig_Cmd_Read.Q THEN
	IN_CmdToggleRead := FALSE;
	MesCP_Read := NOT MesCP_Read;
	
END_IF

IF Trig_Cmd_Write.Q THEN
	IN_CmdToggleWrite := FALSE;
	MesCP_Write := NOT MesCP_Write;
	
END_IF
END_METHOD

METHOD M_Execute : BOOL
VAR_INPUT
END_VAR
	
	TP1(IN:=NOT TP1.Q , PT:= ParamClockRead );
	ClockRead 	:= TP1.Q;
	
	M_CP();
		
	M_Read();
	
	M_Write();
	
	M_AlarmManagement();
END_METHOD

METHOD M_Read : BOOL
VAR_INPUT
END_VAR

VAR
	MW					: FB_MergeWordsToFloat;
END_VAR
END_METHOD

METHOD M_Write : BOOL
VAR
		CmdbyCom	: WORD;
		
END_VAR
END_METHOD

END_FUNCTION_BLOCK

// ---- 01_Equipement_Library/Datalogger/FB_Datalogger_IOWIT.TcPOU
FUNCTION_BLOCK FB_Datalogger_IOWIT EXTENDS FB_Datalogger_Base

VAR_INPUT PERSISTENT
	{attribute 'OPC.UA.DA' := '1'} 
	ParamTcpPort			: UINT   := 502;					(* Modbus TCP port															*)
	{attribute 'OPC.UA.DA' := '1'}                          	
	ParamIPAddress			: STRING;				 			(* (NA)Config: IP Adress of WIT                                             *)
	{attribute 'OPC.UA.DA' := '1'} 	                        	
	ParamUnitID 			: BYTE:=1; 							(* (NA)   SMA Modbus Unit ID.                                               *)
	                                                        	
	ParamTempoComAlarm		: TIME 		:= T#30S ; 				(* (s) Config : Tempo to detect LOC Alarm                                   *)
	ParamTimeOutCurtail     : TIME 		:= T#45S ;				(* (s) Config : Tempo to curtail power at set value before Timeout warning  *)
	ParamClockReadTime 		: TIME 		:= TIME#2S;	  			(* (Time) Read Modbus Frequency .                                           *)
	ParamClockWriteTime 	: TIME 		:= TIME#2S; 	  		(* (Time) Write Modbus Frequency .                                          *)
 	ParamTimeout			: TIME  	:= T#5S ;		  		(* (Time) Timeout for modbus reading                                        *)
		                                                    
	ParamID					: UINT :=1; 						(* ID of the datalogger . Corresponding to PTR ID .                         *)
	
END_VAR

VAR_INPUT 
	// Parameters of the Object (instance specific) 
	IN_CmdToggleRead			: BOOL ;
		
	IN_CmdReset_L				: BOOL ;						// (NA) External Reset Command
	                                                    		
	MbAddrDI	: WORD; 										// Adresse IP Requête Digital Inputs
	MbAddrAI	: ARRAY[1.. 8] OF WORD; 						// Adresses IP Requête Analogic Inputs 
END_VAR

VAR
		
	// M_READ VARIABLES//
MesDataExd AT %Q*			      	: Datalogger_IOWIT ; 	// (NA) [P,H,B] INV  Data Structure 

		
	
	FB_ModbusReadDI	        : FB_ModbusReadCoils;   	 		// FB for Modbus Reading Digital Values
	FB_ModbusReadAI			: FB_ModbusRead;			 		// FB for Modbus Reading Analogic Values (Adresses on 1010X-1019X range)
	
	DI_List : ARRAY[1..27] OF BOOL;
	AI_List : ARRAY[1..18] OF WORD;
	TempAIList : ARRAY[1..2] OF WORD;
		
		
	// M_ALARMMNGMT VARIABLES //
	TON_ComAlarm				: TON ; 						// Tempo before deteting loss of communication. 
	TON_ComWarning				: TON ; 						// Tempo before detecting loss of communication.                                                	
                                 		    	        		
	MesComWarning				: BOOL ; 						// (NA) [P,H]  True if bad communication
                                                        		
	                                                    		
	//M_EXECUTE VARIABLES //                            		
	TP1							: TP ; 	 						// (NA) Tempo to define Modbus Reading Frequency 
	Trig_Cmd_Read: R_TRIG;	                            	
	                                                    	
	ClockRead		AT %Q*		: BOOL	;						// (NA) Modbus reading Clock
    
    
	bInit						: BOOL;
	
	
END_VAR

METHOD M_AlarmManagement
//////////////////
// Manages IntelliGen Alarms
/////////////////

VAR 
	// Method local variables (reinitialized at each cycle) 
	FB_AlarmCodeManager : FB_AlarmCodeManager ; 
	KK				: BYTE;		// For Loop 
	bComError		: BOOL := TRUE;
	bComWarning 	: BOOL;
	AC_CB_OPEN		: BOOL;
END_VAR

// ALARM CODE //
	FB_AlarmCodeManager(
		bAlarm1			:= MesDataExd.MesData.Transfo.MesDataExd.MesData.MesAlarmTemp , 		// A1_Transfo : Temperature alarm
		bAlarm2			:= MesDataExd.MesData.FSS.MesAlarmFire , 					// FSS : Security Fire Detection                                         
		bAlarm3			:= MesDataExd.MesData.Transfo.MesDataExd.MesData.MesAlarmGas ,			// A1_Transfo : Transfo Gaz Discharge                                      
		bAlarm4			:= MesDataExd.MesData.Transfo.MesDataExd.MesData.MesAlarmOilLevel ,	// A1_Transfo : Transfo Pressure 	                                           
		bAlarm5			:= MesDataExd.MesData.MS.MesAlarmState , 					// A1_MS : Security Motion Sensor                                         
		bAlarm6			:= MesDataExd.MesData.DS.MesAlarmState ,					// A1_DS : Security Door Contact                                           
		bAlarm7			:= MesDataExd.MesData.WS.MesSVS_Signal1,					// A1_WS : Security Video Signal 1                                          
		bAlarm8			:= MesDataExd.MesData.WS.MesSVS_Signal2,					// A1_WS : Security Video Signal 2            
		bAlarm9			:= MesDataExd.MesData.WS.MesSVS_Signal3,					// A1_WS : Security Video Signal 3            
		bAlarm10		:= MesDataExd.MesData.CB_Transfo.MesAlarmState, 			// CB_Transfo : Alarm State                                         
		bAlarm11		:= MesDataExd.MesData.CB_INV[1].MesAlarmState, 				// CB_INV_1 : Alarm State                                         
		bAlarm12		:= MesDataExd.MesData.CB_INV[2].MesAlarmState, 				// CB_INV_2 : Alarm State                                         
		bAlarm13		:=FALSE, //                                          
		bAlarm14		:=FALSE, //                                          
		bAlarm15		:=FALSE , 			// 			                                 
		wAlarmCode		=>MesDataExd.MesData.MesAlarmCode);                            

// WARNING CODE //
	FB_AlarmCodeManager(
 		bAlarm1			:= MesDataExd.MesData.Transfo.MesDataExd.MesData.MesWarningTemp,		//	A1_Transfo : Transfo Temp Warning 		
		bAlarm2			:=FALSE, //
		bAlarm3			:=FALSE, //
		bAlarm4			:=FALSE, //                                 
		bAlarm5			:=FALSE, //                          	
		bAlarm6			:=FALSE, //                                   
		bAlarm7			:=FALSE, //                                   
		bAlarm8			:=FALSE, //                                   
		bAlarm9			:=FALSE, //                                   
		bAlarm10		:=FALSE, //                                   
		bAlarm11		:=FALSE, //                                   
		bAlarm12		:=FALSE, //                                   
		bAlarm13		:=FALSE, //                                   
		bAlarm14		:=FALSE, //                                   
		bAlarm15		:=FALSE, //                                   
		wAlarmCode		=>MesDataExd.MesData.MesWarningCode);

// EVENT CODE //
	FB_AlarmCodeManager(
 		bAlarm1			:= MesDataExd.MesData.MesInvReturnContact1, // Inverter Return Contact 1		
		bAlarm2			:= MesDataExd.MesData.MesInvReturnContact2, // Inverter Return Contact 2
		bAlarm3			:=FALSE, //
		bAlarm4			:=FALSE, //                                 
		bAlarm5			:=FALSE, //                          	
		bAlarm6			:=FALSE, //                                   
		bAlarm7			:=FALSE, //                                   
		bAlarm8			:=FALSE, //                                   
		bAlarm9			:=FALSE, //                                   
		bAlarm10		:=FALSE, //                                   
		bAlarm11		:=FALSE, //                                   
		bAlarm12		:=FALSE, //                                   
		bAlarm13		:=FALSE, //                                   
		bAlarm14		:=FALSE, //                                   
		bAlarm15		:=FALSE, //                                   
		wAlarmCode		=>MesDataExd.MesData.MesWarningCode);
END_METHOD

METHOD M_CP
//////////////////
//  Emulator
/////////////////

VAR 
	// Method local variables (reinitialized at each cycle) 
	

END_VAR
Trig_Cmd_Read(CLK:=IN_CmdToggleRead);


IF Trig_Cmd_Read.Q THEN
	IN_CmdToggleRead := FALSE;
MesDataExd.MesData.MesCP_Read := NOT MesDataExd.MesData.MesCP_Read;
END_IF
END_METHOD

METHOD M_Execute
//////////////////
//  Method Calls 
/////////////////

VAR 
	// Method local variables (reinitialized at each cycle) 

END_VAR
M_CP() ; 
M_Read() ; 
M_AlarmManagement() ;
END_METHOD

{attribute 'object_name' := 'M_Read'}
METHOD M_Read
//////////
// Read Method for SMA : Modbus reading
//////////
VAR
	// Method local variables (reinitialized at each cycle) 
	//MW					: FB_MergeWordsToFloat;
	//MW_1				: FB_WordsToDint64BE;
	

	MW					: FB_MergeWordsToDint;
	i 					: INT;
	
	MesInv2SSM6SwitchGear: INT;
	KK: INT;
END_VAR

// CP-Read / Write 

MesDataExd.MesData.MesCP_Read := MesCP_Read ; 
MesDataExd.MesData.MesCP_Write := MesCP_Write ;  

IF MesCP_Read  THEN		 
	
	// Digital Inputs Modbus Requests 
	
	FB_ModbusReadDI(pDestAddr := ADR(DI_List),
					sIPAddr := ParamIPAddress,
					tTimeout := ParamTimeout,
					nTcpPort := 502,
					nQuantity := 28,
					nMBAddr := MbAddrDI,
					cbLength := SIZEOF(DI_List),
					nUnitID := 1,
					ClockRead := MesDataExd.MesData.MesCP_Read AND ClockRead,
					Reset := CmdClearFault_G OR IN_CmdReset_L);
					
	FOR i := 1 TO 8 DO
		FB_ModbusReadAI(pDestAddr := ADR(TempAIList),
					sIPAddr := ParamIPAddress,
					tTimeout := ParamTimeout,
					nTcpPort := 502,
					nQuantity := 2,
					nMBAddr := MbAddrAI[i],
					cbLength := SIZEOF(TempAIList),
					nUnitID := 1,
					ClockRead := MesDataExd.MesData.MesCP_Read AND ClockRead,
					Reset := CmdClearFault_G OR IN_CmdReset_L);
					
		AI_List[2*i-1] := TempAIList[1];
		AI_List[2*i] := TempAIList[2];
	END_FOR	
	
	//  MesDataExd.MesData.Filling Digital Input			
	
	MesDataExd.MesData.MesInvReturnContact1	:=	DI_List[1]; 	
	MesDataExd.MesData.MesInvReturnContact2	:=	DI_List[2]; 
		
	MesDataExd.MesData.Transfo.MesDataExd.MesData.MesAlarmGas 			:= DI_List[3];
	MesDataExd.MesData.Transfo.MesDataExd.MesData.MesAlarmOilLevel 		:= DI_List[4];
	MesDataExd.MesData.Transfo.MesDataExd.MesData.MesWarningTemp 		:= DI_List[5];
	MesDataExd.MesData.Transfo.MesDataExd.MesData.MesAlarmTemp        	:= DI_List[6];
	
	MesDataExd.MesData.CB_Transfo.MesAlarmState	:=	DI_List[7];	// NO ? 
	MesDataExd.MesData.FSS.MesAlarmFire      		:=  DI_List[8];
	 
	MesDataExd.MesData.CB_INV[1].MesAlarmState 	:=	DI_List[9]; 
	MesDataExd.MesData.CB_INV[2].MesAlarmState  	:= 	DI_List[10];
	 
	MesDataExd.MesData.MS.MesAlarmState 	:=	DI_List[11];
	MesDataExd.MesData.DS.MesAlarmState 	:=  DI_List[12];			// MesSecurityDoorContact
	MesDataExd.MesData.WS.MesSVS_Signal1 	:=  DI_List[13];
		
	 FOR KK:= 1 TO CstNbSTR_G DO 
	 	AX_PTR[ParamID].AX_INV[1].MesDataExd.MesData.Fuse_DC[KK].MesAlarmState 	:=	DI_List[14+(KK-1)];		// MesInv1SSM1SwitchGear
	 END_FOR
	  FOR KK:= 1 TO CstNbSTR_G DO 
	 	AX_PTR[ParamID].AX_INV[2].MesDataExd.MesData.Fuse_DC[KK].MesAlarmState 	:=	DI_List[20+(KK-1)];		// MesInv1SSM1SwitchGear
	 END_FOR
	 
	
	MesDataExd.MesData.WS.MesSVS_Signal2	:=	DI_List[26];
	MesDataExd.MesData.WS.MesSVS_Signal3 :=  DI_List[27];
	 
	 
	 
	 (*
	MesDataExd.MesData.MesInvReturnContact1	:=	DI_List[1]; 	
	MesDataExd.MesData.MesInvReturnContact2	:=	DI_List[2]; 
		
	MesDataExd.MesData.MesTransfoGazDischarge		:= DI_List[3];
	MesDataExd.MesData.MesTransfoPressure		   	:= DI_List[4];
	MesDataExd.MesData.MesTransfoTempWarning		:= DI_List[5];
	MesDataExd.MesData.MesTransfoTempTrig        	:= DI_List[6];
	
	MesDataExd.MesData.MesHVAuxSwitchGearTransfo	:=	DI_List[7];
	MesDataExd.MesData.MesSecurityFireDetect     	:=  DI_List[8];
	 
	MesDataExd.MesData.MesHVAuxSwitchGearInv1	:=	DI_List[9]; 
	MesDataExd.MesData.MesHVAuxSwitchGearInv2  := 	DI_List[10];
	 
	MesDataExd.MesData.MesSecurityMotionSensor	:=	DI_List[11];
	MesDataExd.MesData.MesSecurityDoorContact	:=  DI_List[12];
	MesDataExd.MesData.A1_WS.MesSVS_Signal1 :=  DI_List[13];
		
	MesDataExd.MesData.MesInv1SSM1SwitchGear	:=	DI_List[14];
	MesDataExd.MesData.MesInv1SSM2SwitchGear	:=	DI_List[15];
	MesDataExd.MesData.MesInv1SSM3SwitchGear   :=  DI_List[16];
	MesDataExd.MesData.MesInv1SSM4SwitchGear	:=  DI_List[17];
	MesDataExd.MesData.MesInv1SSM5SwitchGear   :=  DI_List[18];
	MesDataExd.MesData.MesInv1SSM6SwitchGear	:=  DI_List[19];
	MesDataExd.MesData.MesInv2SSM1SwitchGear   :=  DI_List[20];
	MesDataExd.MesData.MesInv2SSM2SwitchGear   :=  DI_List[21];
	MesDataExd.MesData.MesInv2SSM3SwitchGear   :=  DI_List[22];
	MesDataExd.MesData.MesInv2SSM4SwitchGear   :=  DI_List[23];
	MesDataExd.MesData.MesInv2SSM5SwitchGear   :=  DI_List[24];
	MesDataExd.MesData.MesInv2SSM6SwitchGear   :=  DI_List[25];
	*)
	
	
	//  MesDataExd.MesData.Filling Analogic Input
	
	
	MW(WORD_STRONG :=  AI_List[1],	WORD_WEAK := AI_List[2], SIZE := 1, FIX := 0, SIGNED := 0, VAR_OUT	:= MesDataExd.MesData.MesTransfoLocalTemp);
	MW(WORD_STRONG :=  AI_List[3],	WORD_WEAK := AI_List[4], SIZE := 1, FIX := 0, SIGNED := 0, VAR_OUT	:= MesDataExd.MesData.WS.MesTempMod1);
	MW(WORD_STRONG :=  AI_List[5],	WORD_WEAK := AI_List[6], SIZE := 1, FIX := 0, SIGNED := 0, VAR_OUT	:= MesDataExd.MesData.WS.MesTempMod2);
	MW(WORD_STRONG :=  AI_List[7],	WORD_WEAK := AI_List[8], SIZE := 1, FIX := 0, SIGNED := 0, VAR_OUT	:= MesDataExd.MesData.WS.MesTempExt);
	MW(WORD_STRONG :=  AI_List[9],	WORD_WEAK := AI_List[10], SIZE := 1, FIX := 0, SIGNED := 0, VAR_OUT	:= MesDataExd.MesData.WS.MesWindSpd);		
	MW(WORD_STRONG :=  AI_List[11],	WORD_WEAK := AI_List[12], SIZE := 1, FIX := 0, SIGNED := 0, VAR_OUT	:= MesDataExd.MesData.WS.MesGHI_Left);	  
	MW(WORD_STRONG :=  AI_List[13],	WORD_WEAK := AI_List[14], SIZE := 1, FIX := 0, SIGNED := 0, VAR_OUT	:= MesDataExd.MesData.WS.MesGHI_Middle);	
	MW(WORD_STRONG :=  AI_List[15],	WORD_WEAK := AI_List[16], SIZE := 1, FIX := 0, SIGNED := 0, VAR_OUT	:= MesDataExd.MesData.WS.MesGHI_Right);	 
	
END_IF
END_METHOD

END_FUNCTION_BLOCK

// ---- 01_Equipement_Library/Datalogger/FB_Datalogger_SchSkid.TcPOU
FUNCTION_BLOCK FB_Datalogger_SchSkid EXTENDS FB_Datalogger_Base
 

VAR_INPUT PERSISTENT
	ParamID_PTR					: BYTE; 				 						(* (NA) ID of the datalogger. Corresponding to PTR ID *)
	ParamWriteTimeout			: TIME  	:= T#5S ;		  					(* (Time) Timeout for modbus reading*)
END_VAR

       	
VAR_INPUT           	
	// I/O Inputs 
	
END_VAR             	
      	
VAR                 	
MesDataExd  AT %Q*		: Datalogger_SchSkid;

	CmdbyCom 		AT %Q*		: WORD;
	
//INPUT Modbus
	FB_ModbusRead	          	: ARRAY[1..2] OF FB_ModbusRead; 	            // (NA) FB for Modbus Reading
	FB_COMWrite					: FB_ModbusWrite;
	MesBlock1_Temp				: ARRAY [1..19] OF WORD ; 
	MesBlock2_Temp 				: ARRAY [1..26] OF WORD ; 
	
	ModbusInputBoolAlarms		: BOOL;
	ModbusInputBoolAlarmId		: UDINT;
	ModbusInputAnaAlarms		: BOOL;
	ModbusInputAnaAlarmId		: UDINT;
	TEMP_4_20					: ARRAY [1..13] OF REAL;

//OUTPUT Modbus
	MesModbusCmdByComAlarm 		: BOOL;
	MesModbusCmdByComCodeId		: UDINT;
	Front_Montant				: R_Trig;
	RS_Open						: RS;
	RS_Close					: RS;
	
END_VAR

METHOD M_AlarmManagement
//////////////////
// Generates object alarms and manages resets. 
//////////////////

VAR 
	// Method local variables (reinitialized at each cycle) 
	FB_AlarmCodeManager		: FB_AlarmCodeManager;  
END_VAR
	
// ALARM CODE //
	FB_AlarmCodeManager(
		bAlarm1				:= MesDataExd.Transfo_Synthesis.MesData.MesAlarmsSynthesis,		// Synthesis : trip of DGPT2 ON G,P,T (from DI_208)
		bAlarm2				:= MesDataExd.Transfo_Synthesis.MesData.MesAlarmTemp,			// Synthesis : alarms temperature (from DI_207) 
		bAlarm3				:= MesDataExd.DS_Synthesis.MesAlarmState,						// Synthesis : door positions (from DI_209)
		bAlarm4				:= FALSE,														//
		bAlarm5				:= FALSE,														//
		bAlarm6				:= FALSE,														//
		bAlarm7				:= FALSE,														//
		bAlarm8				:= FALSE,														//
		bAlarm9				:= FALSE,														//
		bAlarm10			:= FALSE,														//
		bAlarm11			:= MesDataExd.CB_INV[1].MesAlarmState, 							// CB_INV_1 : alarm state 
		bAlarm12			:= MesDataExd.CB_INV[2].MesAlarmState, 							// CB_INV_2 : alarm state 
		bAlarm13			:= FALSE, 														//                                          
		bAlarm14			:= FALSE,														//                                          
		bAlarm15			:= FALSE,														// 		
		wAlarmCode			=>MesDataExd.MesData.MesAlarmCode);										//
			
// WARNING CODE //
	FB_AlarmCodeManager(
		bAlarm1				:= FALSE, 														// 
		bAlarm2				:= FALSE, 														//
		bAlarm3				:= FALSE,														//
		bAlarm4				:= FALSE,														//
		bAlarm5				:= FALSE,														//
		bAlarm6				:= FALSE,														//
		bAlarm7				:= FALSE,														//
		bAlarm8				:= FALSE,														//
		bAlarm9				:= FALSE,														//
		bAlarm10			:= FALSE,														//
		bAlarm11			:= FALSE,														//
		bAlarm12			:= FALSE,														//
		bAlarm13			:= FALSE,														//
		bAlarm14			:= FALSE,														//
		bAlarm15			:= FALSE,														//
		wAlarmCode			=>MesDataExd.MesData.MesWarningCode);										//
		                                                        							
// EVENT CODE //                                                							
                                                                							
	FB_AlarmCodeManager(                                        							
		bAlarm1				:= FALSE,						    							//  
		bAlarm2				:= FALSE, 														//  
		bAlarm3				:= FALSE,														//
		bAlarm4				:= FALSE,														//
		bAlarm5				:= FALSE,														//
		bAlarm6				:= FALSE,														//
		bAlarm7				:= FALSE,														//
		bAlarm8				:= FALSE,														//
		bAlarm9				:= FALSE,														//
		bAlarm10			:= FALSE,														//
		bAlarm11			:= FALSE,														//
		bAlarm12			:= FALSE,														//
		bAlarm13			:= FALSE,														//
		bAlarm14			:= FALSE,														//
		bAlarm15			:= FALSE,														//
		wAlarmCode			=>MesDataExd.MesData.MesEventCode);										//
END_METHOD

METHOD M_CP

VAR 
	// Method local variables (reinitialized at each cycle) 
	
END_VAR
SUPER^.M_CP() ;
END_METHOD

METHOD M_Execute : BOOL
VAR_INPUT
END_VAR
IF bInit THEN
	M_Init();
	bInit := FALSE;
ELSIF CmdInit_G THEN 
	bInit:= TRUE ;
END_IF

SUPER^.M_Execute() ;
END_METHOD

METHOD M_Init : BOOL
VAR_INPUT
END_VAR
END_METHOD


METHOD M_Read : BOOL
VAR_INPUT
END_VAR

VAR
	MW					: FB_MergeWordsToFloat;
END_VAR
// CP-Read / Write 

MesDataExd.MesData.MesCP_Read := MesCP_Read ; 
MesDataExd.MesData.MesCP_Write := MesCP_Write ;  

IF MesCP_Read  THEN	
//DI MODBUS	
	FB_ModbusRead[1]
		(
			nTCPPort		:= ParamTcpPort,
			ClockRead		:= MesCP_Read AND ClockRead, 
			Reset			:= CmdClearFault_G OR IN_CmdReset_L,
			sIPAddr			:= ParamIPAddress ,
			nUnitID			:= 1, 
			tTimeout		:= T#5S,
			nQuantity		:= 19, 
			nMBAddr			:= 300 , 
			cbLength		:= SIZEOF(MesBlock1_Temp), 
			pDestAddr		:= ADR(MesBlock1_Temp), 
			ModbusReadAlarm	=> ModbusInputBoolAlarms, 
			ErrorId			=> ModbusInputBoolAlarmId
		);
//4-20ma MODBUS	
		FB_ModbusRead[2]
		(
			nTCPPort		:= ParamTcpPort,
			ClockRead		:= MesCP_Read AND ClockRead, 
			Reset			:= CmdClearFault_G OR IN_CmdReset_L,
			sIPAddr			:= ParamIPAddress ,
			nUnitID			:= 1, 
			tTimeout		:= T#5S,
			nQuantity		:= 26, 
			nMBAddr			:= 400 , 
			cbLength		:= SIZEOF(MesBlock2_Temp), 
			pDestAddr		:= ADR(MesBlock2_Temp), 
			ModbusReadAlarm	=> ModbusInputAnaAlarms, 
			ErrorId			=> ModbusInputAnaAlarmId
		);

	
//DI	
MesDataExd.MesWatchdog_ProtectRelayVIP 						:= WORD_TO_BOOL(MesBlock1_Temp[1]);
MesDataExd.CB_INV[1].MesAlarmState							:= WORD_TO_BOOL(MesBlock1_Temp[2]);
MesDataExd.CB_INV[2].MesAlarmState							:= WORD_TO_BOOL(MesBlock1_Temp[3]); 
MesDataExd.MesComutLocal									:= WORD_TO_BOOL(MesBlock1_Temp[4]);
MesDataExd.MesState_MVCB									:= WORD_TO_BOOL(MesBlock1_Temp[5]);
MesDataExd.MesFault_ProtectRelayVIP							:= WORD_TO_BOOL(MesBlock1_Temp[6]);
MesDataExd.Transfo_Synthesis.MesData.MesAlarmTemp			:= WORD_TO_BOOL(MesBlock1_Temp[7]);
MesDataExd.Transfo_Synthesis.MesData.MesAlarmsSynthesis		:= WORD_TO_BOOL(MesBlock1_Temp[8]);
MesDataExd.DS_Synthesis.MesAlarmState						:= WORD_TO_BOOL(MesBlock1_Temp[9]); 				// TRUE OUVERT
	
	IF 	ParamID_PTR	= 4 THEN
	MesDataExd.CB_INV[1].MesAlarmState 						:= MesDataExd.CB_INV[2].MesAlarmState; 				// CB of inverter one is in inverter 2
	END_IF	
	
//4-20ma
	MW( WORD_STRONG:= MesBlock2_Temp[2  ],	WORD_WEAK := MesBlock2_Temp[1  ], VAR_OUT :=Temp_4_20[1] ); 		//
    MW( WORD_STRONG:= MesBlock2_Temp[4  ], 	WORD_WEAK := MesBlock2_Temp[3  ], VAR_OUT :=Temp_4_20[2] ); 		// 
    MW( WORD_STRONG:= MesBlock2_Temp[6  ], 	WORD_WEAK := MesBlock2_Temp[5  ], VAR_OUT :=Temp_4_20[3] ); 		// 
    MW( WORD_STRONG:= MesBlock2_Temp[8  ], 	WORD_WEAK := MesBlock2_Temp[7  ], VAR_OUT :=Temp_4_20[4] ); 		// 
    MW( WORD_STRONG:= MesBlock2_Temp[10 ], 	WORD_WEAK := MesBlock2_Temp[9  ], VAR_OUT :=Temp_4_20[5] );		// 
    MW( WORD_STRONG:= MesBlock2_Temp[12 ], 	WORD_WEAK := MesBlock2_Temp[11 ], VAR_OUT :=Temp_4_20[6] );  
    MW( WORD_STRONG:= MesBlock2_Temp[14 ], 	WORD_WEAK := MesBlock2_Temp[13 ], VAR_OUT :=Temp_4_20[7] );		// Pyrano route PTR1,2,4 / wind speed for PTR3
    MW( WORD_STRONG:= MesBlock2_Temp[16 ], 	WORD_WEAK := MesBlock2_Temp[15 ], VAR_OUT :=Temp_4_20[8] ); 		// Pyrano eau PTR1,2,4 / wind direction for PTR3
    MW( WORD_STRONG:= MesBlock2_Temp[18 ], 	WORD_WEAK := MesBlock2_Temp[17 ], VAR_OUT :=Temp_4_20[9] ); 		// Temp panel
    MW( WORD_STRONG:= MesBlock2_Temp[20 ], 	WORD_WEAK := MesBlock2_Temp[19 ], VAR_OUT :=Temp_4_20[10]); 
    MW( WORD_STRONG:= MesBlock2_Temp[22 ], 	WORD_WEAK := MesBlock2_Temp[21 ], VAR_OUT :=Temp_4_20[11]); 
    //MW( WORD_STRONG_F:= MesBlock2_Temp[24 ], 	WORD_WEAK_F := MesBlock2_Temp[23 ], NUMBER_F := MesDataExd.MesData.MesTemp_TrasfoOil_1  ); // Tp Transfo 1
	//MW( WORD_STRONG_F:= MesBlock2_Temp[26 ], 	WORD_WEAK_F := MesBlock2_Temp[25 ], NUMBER_F := MesDataExd.MesData.MesTemp_TrasfoOil_2  ); // Tp Transfo 2
END_IF
END_METHOD

METHOD M_Write : BOOL
VAR
		
		
END_VAR
IF AX_PTR[ParamID_PTR].A1_MainMVCB_PTR.OUT_CmdClose_IO THEN
	CmdbyCom.0 := 0;
	CmdbyCom.1 := 1;
END_IF
	
IF AX_PTR[ParamID_PTR].A1_MainMVCB_PTR.OUT_CmdOpen_IO THEN
	CmdbyCom.0 := 1;
	CmdbyCom.1 := 0;
END_IF

Front_Montant(CLK:= AX_PTR[ParamID_PTR].A1_MainMVCB_PTR.OUT_CmdClose_IO OR AX_PTR[ParamID_PTR].A1_MainMVCB_PTR.OUT_CmdOpen_IO);
RS_Open(SET:=Front_Montant.Q,Reset1:= NOT MesDataExd.MesState_MVCB OR IN_CmdReset_L );

RS_Close(SET:=Front_Montant.Q,Reset1:=MesDataExd.MesState_MVCB OR IN_CmdReset_L);


FB_COMWrite(
		pSrcAddr 			:= ADR(CmdbyCom) ,
		cbLength			:= SIZEOF(CmdbyCom) , 
		nQuantity 			:= 1,
		Reset				:= CmdClearFault_G OR IN_CmdReset_L, 
		sIPAddr				:= ParamIPAddress , 
		nUnitID				:= 1 , //modif LWN
		nMBAddr				:= 40302 , 
		tTimeout			:= ParamWriteTimeout ,
		WriteCmd			:= (RS_Open.Q1 OR RS_close.Q1) and MesCP_Write, 
		ModbusWriteAlarm	=> MesModbusCmdByComAlarm , 
		ErrorId				=> MesModbusCmdByComCodeId);
END_METHOD

END_FUNCTION_BLOCK

// ---- 01_Equipement_Library/Datalogger/FB_Datalogger_SENECA.TcPOU
FUNCTION_BLOCK FB_Datalogger_SENECA EXTENDS FB_Datalogger_Base
 

VAR_INPUT PERSISTENT
	ParamWriteTimeout			: TIME  	:= T#5S ;		  					(* (Time) Timeout for modbus reading*)
END_VAR

       	
VAR_INPUT           	
	// I/O Inputs 
	
END_VAR             	
      	
